(* CODESYS project NETWORK.library
   Author: OSCAT
   Version: 1.3.5.1
   Description: Oscat Network Version 07/2017 aus *.lib
      Formale Korrekturen von annD und Referenzen "Variabeln LOC_DT et.al." für Kompatibilität mit Codesys 3.5.16.0 angepasst
   Title: NETWORK
   Placeholder: OSCAT_NETWORK
   DefaultNamespace: OSCAT_NETWORK
   Company: OSCAT

Project tree, tasks and I/O mapping:
  libraries: IecSfc, 3.4.2.0 (System); Analyzation, 3.5.15.0 (System); Standard, 3.5.15.0 (System); BASIC, 3.5.16.0 (OSCAT); SysFile, 3.5.15.0 (System); SysSocket, 3.5.15.0 (System); SysSocket2, 3.5.16.10 (System); SysTypes Interfaces, 3.5.2.0 (System)
  Data types/
    DATA_LOG/
      data type DLOG_CRON_DATA
      data type DLOG_CRON_ELEMENT
      data type DLOG_DATA
      data type DLOG_REAL_ARRAY_DATA
      data type DLOG_REAL_ARRAY_ELEMENT
      data type DLOG_RETAIN
      data type DLOG_SAVE
      data type LOG_CONTROL
      data type PRINTF_DATA
      data type UNI_CIRCULAR_BUF
      data type UNI_CIRCULAR_BUFFER_DATA
      data type us_LOG_VIEWPORT
    DATABASE/
      data type MYSQL_COM
      data type MYSQL_INFO
    FILE_SERVER/
      data type FILE_PATH_DATA
      data type FILE_SERVER_DATA
      data type FILE_SERVER_RUNTIME_DATA
    NET_VAR/
      data type NET_VAR_DATA
    NETWORK/
      data type IP2GEO_DATA
      data type IP_C
      data type IP_FIFO_DATA
      data type NETWORK_BUFFER
      data type NETWORK_BUFFER_SHORT
      data type NW_BUF_LONG
      data type NW_BUF_SHORT
      data type URL
      data type VMAP_DATA
      data type XML_CONTROL
    TELNET_VISION/
      data type us_TN_INPUT_CONTROL
      data type us_TN_INPUT_CONTROL_DATA
      data type us_TN_MENU
      data type us_TN_MENU_POPUP
      data type us_TN_SCREEN
    WEATHER/
      data type WORLD_WEATHER_CUR
      data type WORLD_WEATHER_DATA
      data type WORLD_WEATHER_DAY
      data type YAHOO_WEATHER_DATA
      data type YAHOO_WEATHER_FORECAST_DAY
  Global Variables/
    global variables Constants
    global variables Globale_Variablen
  POUs/
    CONVERT/
      function block BASE64_DECODE_STR [ST]
      function block BASE64_DECODE_STREAM [ST]
      function block BASE64_ENCODE_STR [ST]
      function block BASE64_ENCODE_STREAM [ST]
      function HTML_DECODE [ST]
      function HTML_ENCODE [ST]
      function IP4_CHECK [ST]
      function IP4_DECODE [ST]
      function IP4_TO_STRING [ST]
      function IS_IP4 [ST]
      function IS_URLCHR [ST]
      function MD5_AUX [ST]
      function block MD5_CRAM_AUTH [ST]
      function block MD5_STR [ST]
      function block MD5_STREAM [ST]
      function MD5_TO_STRH [ST]
      function block RC4_CRYPT_STREAM [ST]
      function block SHA1_STR [ST]
      function block SHA1_STREAM [ST]
      function SHA1_TO_STRH [ST]
      function STRING_TO_URL [ST]
      function URL_DECODE [ST]
      function URL_ENCODE [ST]
      function URL_TO_STRING [ST]
    DATA_LOG/
      function block DLOG_BOOL [ST]
      function block DLOG_CRON_TAB [ST]
      function block DLOG_DINT [ST]
      function block DLOG_DT [ST]
      function block DLOG_FILE_TO_FTP [ST]
      function block DLOG_FILE_TO_SMTP [ST]
      function block DLOG_REAL [ST]
      function block DLOG_REAL_ARRAY [ST]
      function block DLOG_STORE_FILE_CSV [ST]
      function block DLOG_STORE_FILE_HTML [ST]
      function block DLOG_STORE_FILE_XML [ST]
      function block DLOG_STORE_MYSQL [ST]
      function block DLOG_STORE_RRD [ST]
      function block DLOG_STRING [ST]
    DATABASE/
      function block MYSQL_AUTH [ST]
      function block MYSQL_CONTROL [ST]
    DEMO/
      program BASE64_DEMO [CFC]
      program CSV_PARSER_BUF_DEMO [ST]
      program CSV_PARSER_FILE_DEMO [ST]
      program DLOG_FILE_CSV_DEMO [CFC]
      program DLOG_FILE_CSV_FTP_DEMO [CFC]
      program DLOG_FILE_CSV_SMTP_DEMO [CFC]
      program DLOG_FILE_HTML_DEMO [CFC]
      program DLOG_FILE_XML_DEMO [CFC]
      program DLOG_MYSQL_DEMO [CFC]
      program DLOG_RRD_DEMO [CFC]
      program DNS_DYN_DEMO [CFC]
      program DNS_REV_DEMO [CFC]
      program DNS_SNTP_SYSLOG_DEMO [CFC]
      program FILE_BLOCK_DEMO [CFC]
      program FTP_CLIENT_DEMO [CFC]
      program GET_WAN_IP_DEMO [CFC]
      program HTTP_DEMO [CFC]
      program INI_PARSER_BUF_DEMO [ST]
      program INI_PARSER_FILE_DEMO [ST]
      program IP2GEO_DEMO [CFC]
      program IRTRANS_DEMO [CFC]
      program MB_CLIENT_DEMO [CFC]
      program MB_SERVER_DEMO [CFC]
      program MD5_CRAM_AUTH_DEMO [CFC]
      program NET_VAR_MASTER_DEMO [CFC]
      program NET_VAR_SLAVE_DEMO [CFC]
      program RC4_CRYPT_DEMO [CFC]
      program SHA1_MD5_DEMO [CFC]
      program SMTP_CLIENT_DEMO [CFC]
      program SPIDER_DEMO [CFC]
      program TELNET_LOG_DEMO [CFC]
      program TELNET_PRINT_DEMO [CFC]
      program TN_VISION_DEMO_1 [ST]
      program TN_VISION_DEMO_2 [ST]
      program WORLD_WEATHER_DEMO [CFC]
      program YAHOO_WEATHER_DEMO [CFC]
    DRIVER/
      function block IRTRANS_DECODE [ST]
      function block IRTRANS_RCV_1 [ST]
      function block IRTRANS_RCV_4 [ST]
      function block IRTRANS_RCV_8 [ST]
      function block IRTRANS_SERVER [ST]
      function block IRTRANS_SND_1 [ST]
      function block IRTRANS_SND_4 [ST]
      function block IRTRANS_SND_8 [ST]
    FILE/
      function block CSV_PARSER_BUF [ST]
      function block CSV_PARSER_FILE [ST]
      function block FILE_BLOCK [ST]
      function FILE_PATH_SPLIT [ST]
      function block INI_PARSER_BUF [ST]
      function block INI_PARSER_FILE [ST]
    HARDWARE/
      function block FILE_SERVER [ST]
      function block FILE_SERVER_RUNTIME [ST]
      function block IP_CONTROL2 [ST]
      function block IP_CONTROL [ST]
    NET_VAR/
      function block NET_VAR_BOOL8 [ST]
      function block NET_VAR_BUFFER [ST]
      function block NET_VAR_CONTROL [ST]
      function block NET_VAR_DWORD8 [ST]
      function block NET_VAR_REAL8 [ST]
      function block NET_VAR_STRING [ST]
      function block NET_VAR_X8 [ST]
    NETWORK/
      function block DNS_CLIENT [ST]
      function block DNS_DYN [ST]
      function block DNS_REV_CLIENT [ST]
      function block FTP_CLIENT [ST]
      function block GET_WAN_IP [ST]
      function block HTTP_GET [ST]
      function block IP2GEO [ST]
      function block MB_CLIENT [ST]
      function block MB_SERVER [ST]
      function block MB_SERVER_1 [ST]
      function block MB_VMAP [ST]
      function block READ_HTTP [ST]
      function block SMTP_CLIENT [ST]
      function block SNTP_CLIENT [ST]
      function block SNTP_SERVER [ST]
      function block SPIDER_ACCESS [ST]
      function block SYS_LOG [ST]
      function block TELNET_LOG [ST]
      function block TELNET_PRINT [ST]
    OTHER/
      function ELEMENT_COUNT [ST]
      function ELEMENT_GET [ST]
      function block IP_FIFO [ST]
      function block LOG_MSG [ST]
      function block LOG_VIEWPORT [ST]
      function NETWORK_VERSION [ST]
      function block PRINT_SF [ST]
      function block UNI_CIRCULAR_BUFFER [ST]
      function block XML_READER [ST]
    TELNET_VISION/
      function block TN_FRAMEWORK [ST]
      function block TN_INPUT_CONTROL [ST]
      function block TN_INPUT_EDIT_LINE [ST]
      function block TN_INPUT_MENU_BAR [ST]
      function block TN_INPUT_MENU_POPUP [ST]
      function block TN_INPUT_SELECT_POPUP [ST]
      function block TN_INPUT_SELECT_TEXT [ST]
      function block TN_RECEIVE [ST]
      function block TN_SC_ADD_SHADOW [ST]
      function block TN_SC_AREA_RESTORE [ST]
      function block TN_SC_AREA_SAVE [ST]
      function block TN_SC_BOX [ST]
      function block TN_SC_FILL [ST]
      function block TN_SC_LINE [ST]
      function block TN_SC_READ_ATTR [ST]
      function block TN_SC_READ_CHAR [ST]
      function TN_SC_SHADOW_ATTR [ST]
      function block TN_SC_VIEWPORT [ST]
      function block TN_SC_WRITE [ST]
      function block TN_SC_WRITE_ATTR [ST]
      function block TN_SC_WRITE_C [ST]
      function block TN_SC_WRITE_CHAR [ST]
      function block TN_SC_WRITE_EOS [ST]
      function TN_SC_XY2_ERROR [ST]
      function TN_SC_XY_ERROR [ST]
      function block TN_SEND_ROWS [ST]
    WEATHER/
      function block MOON_PHASE [ST]
      function block WORLD_WEATHER [ST]
      function block WORLD_WEATHER_DESC_GE [ST]
      function block WORLD_WEATHER_ICON_OSCAT [ST]
      function block YAHOO_WEATHER [ST]
      function block YAHOO_WEATHER_DESC_GE [ST]
      function block YAHOO_WEATHER_ICON_OSCAT [ST]
*)

// Data types/DATA_LOG/DLOG_CRON_DATA
TYPE DLOG_CRON_DATA :
STRUCT
	CE : ARRAY [0..5] OF DLOG_CRON_ELEMENT;
END_STRUCT
END_TYPE

// Data types/DATA_LOG/DLOG_CRON_ELEMENT
TYPE DLOG_CRON_ELEMENT :
STRUCT
	ELEMENTS : ARRAY [0..59] OF BOOL;
	VALUE : INT;
	VALUE_MIN : INT;
	VALUE_MAX : INT;
	ALL_SELECTED : BOOL;
END_STRUCT
END_TYPE

// Data types/DATA_LOG/DLOG_DATA
TYPE DLOG_DATA :
STRUCT
	STORE_TYPE : BYTE;
	ADD_COM : INT;
	ADD_DATA_REQ : BOOL;
	CLOCK_TRIG : BOOL;
	ID_MAX : USINT;
	DTI : DT;
	UCB : UNI_CIRCULAR_BUFFER_DATA;
	LOAD_TIME_MAX : TIME;
	NEW_FILE : STRING;
	NEW_FILE_SIZE : UDINT;
	NEW_FILE_RTRIG : BOOL;
END_STRUCT
END_TYPE

// Data types/DATA_LOG/DLOG_REAL_ARRAY_DATA
TYPE
	DLOG_REAL_ARRAY_DATA : ARRAY [1..64] OF DLOG_REAL_ARRAY_ELEMENT;
END_TYPE

// Data types/DATA_LOG/DLOG_REAL_ARRAY_ELEMENT
TYPE DLOG_REAL_ARRAY_ELEMENT :
STRUCT
	VALUE : REAL;
	DELTA : REAL;
	COLUMN : STRING(10);
	_DELTA_LAST : 	REAL;
	_VALUE_LAST : 	REAL;
END_STRUCT
END_TYPE

// Data types/DATA_LOG/DLOG_RETAIN
TYPE DLOG_RETAIN :
STRUCT
	FN_REM : STRING;
	COLOR : BOOL;
	HEAD: BOOL;
	TRIG_CNT : UDINT;
	TRIG_CNT_TOTAL : UDINT;
END_STRUCT
END_TYPE

// Data types/DATA_LOG/DLOG_SAVE
TYPE DLOG_SAVE :
STRUCT
	FN_REM : STRING;
	COLOR : BOOL;
	HEAD: BOOL;
	TRIG_CNT : UDINT;
	TRIG_CNT_TOTAL : UDINT;
END_STRUCT
END_TYPE

// Data types/FILE_SERVER/FILE_PATH_DATA
TYPE FILE_PATH_DATA :
STRUCT
	DRIVE : STRING(3);
	DIRECTORY : STRING(OSCAT_BASIC.STRING_LENGTH);
	FILENAME : STRING;
END_STRUCT
END_TYPE

// Data types/FILE_SERVER/FILE_SERVER_DATA
TYPE FILE_SERVER_DATA :
STRUCT
	FILE_OPEN : BOOL;
	FILENAME : STRING;
	MODE : BYTE;
	OFFSET : UDINT;
	FILE_SIZE : UDINT;
	ERROR : BYTE;
	RUNTIME : FILE_SERVER_RUNTIME_DATA;
END_STRUCT
END_TYPE

// Data types/FILE_SERVER/FILE_SERVER_RUNTIME_DATA
TYPE FILE_SERVER_RUNTIME_DATA :
STRUCT
	TIME_FILE_OPEN_CUR : UDINT;
	TIME_FILE_OPEN_MAX : UDINT;
	TIME_FILE_OPEN_MIN : UDINT;
	TIME_FILE_CLOSE_CUR : UDINT;
	TIME_FILE_CLOSE_MAX : UDINT;
	TIME_FILE_CLOSE_MIN : UDINT;
	TIME_FILE_READ_CUR: UDINT;
	TIME_FILE_READ_MAX : UDINT;
	TIME_FILE_READ_MIN : UDINT;
	TIME_FILE_WRITE_CUR : UDINT;
	TIME_FILE_WRITE_MAX : UDINT;
	TIME_FILE_WRITE_MIN : UDINT;
	TIME_FILE_SEEK_CUR : UDINT;
	TIME_FILE_SEEK_MAX : UDINT;
	TIME_FILE_SEEK_MIN : UDINT;
	TIME_FILE_TELL_CUR : UDINT;
	TIME_FILE_TELL_MAX : UDINT;
	TIME_FILE_TELL_MIN : UDINT;
	TIME_FILE_DELETE_CUR : UDINT;
	TIME_FILE_DELETE_MAX : UDINT;
	TIME_FILE_DELETE_MIN : UDINT;
END_STRUCT
END_TYPE

// Data types/NETWORK/IP2GEO_DATA
TYPE IP2GEO_DATA :
STRUCT
	STATE : BOOL;
	IP4 : DWORD;
	COUNTRY_CODE : STRING(2);
	COUNTRY_NAME : STRING(20);
	REGION_CODE : STRING(2);
	REGION_NAME : STRING(20);
	CITY : STRING(20);
	GEO_LATITUDE : REAL;
	GEO_LONGITUDE : REAL;
	TIME_ZONE_NAME : STRING(20);
	GMT_OFFSET : INT;
	IS_DST : BOOL;
END_STRUCT
END_TYPE

// Data types/NETWORK/IP_C
TYPE IP_C :
STRUCT
	C_MODE : BYTE;						(*W Mode: TCP/UCP AKTIV/PASSIV                               *)
	C_PORT : WORD;						(*W Portnummer                                               *)
	C_IP : DWORD;						(*W IP-Adresse gepackt wwxxyyzz = www.xxx.yyy.zzz            *)
	C_STATE : BYTE;						(*R Verbindungsstatus ON/OFF + Flanke ON/OFF                 *)
	C_ENABLE : BOOL;					(*W Freigabe für Connect                                     *)
	R_OBSERVE : BOOL;					(*W Empfang ueberwachen                                      *)
	TIME_RESET : BOOL;					(*W Alle Timer ruecksetzen                                   *)
	ERROR : DWORD;					(*R vvwwxxyy (vv = CON_ERROR, ww = SEN_ERROR, xx = REC_ERROR *)
	FIFO : IP_FIFO_DATA;					(*I IP FIFO Struktur                                         *)
	MAILBOX : ARRAY [1..16] OF BYTE;	(*I Mailbox: Datenbereich für Bausteindatenaustausch         *)
	ResultSend:RTS_IEC_RESULT; 			(*Result of TCP Send call*)
	ResultReceive:RTS_IEC_RESULT;		(*Result of TCP Receive call*)
END_STRUCT
END_TYPE

// Data types/NETWORK/IP_FIFO_DATA
TYPE IP_FIFO_DATA :
STRUCT
	X : ARRAY [1..128] OF BYTE; 	(* IP_ID FIFO Speicher          *)
	Y : ARRAY [1..128] OF BYTE; 	(* IP_ID Zähler                 *)
	ID : BYTE;					(* höchste vergabene id         *)
	MAX_ID : BYTE;				(* maximal Anmeldungen pro ID   *)
	INIT : BOOL;					(* Initialisierung durchgeführt *)
	EMPTY : BOOL;				(* FIFO leer                    *)
	FULL : BOOL;					(* FIFO voll                    *)
	TOP : INT;					(* maximale anzahl in FIFO      *)
	NW : INT;					(* Schreibzeiger                *)
	NR : INT;						(* Lesezeiger                   *)
END_STRUCT
END_TYPE

// Data types/DATA_LOG/LOG_CONTROL
TYPE LOG_CONTROL :
STRUCT
	NEW_MSG : STRING(LOG_SIZE); (* neue Nachricht für den Datenbuffer *)
	NEW_MSG_OPTION : DWORD;
	LEVEL : BYTE;
	SIZE : INT := LOG_MAX; (* Anzahl der Strings im LOG_DATA *)
	RESET : BOOL; (* Nachrichtenbuffer löschen *)
	PRINTF : PRINTF_DATA; (* Array PRINTF Parameter *)
	MSG : ARRAY [0..LOG_MAX] OF STRING(LOG_SIZE); (* Array Message *)
	MSG_OPTION : ARRAY [0..LOG_MAX] OF DWORD; (* Array Options *)
	UPDATE_COUNT : UINT; (* Updatezähler *)
	IDX : INT; (* aktueller Nachrichten-Index *)
	RING_MODE : BOOL; (* Bufferüberlauf erkannt *)
END_STRUCT
END_TYPE

// Data types/DATABASE/MYSQL_COM
TYPE MYSQL_COM :
STRUCT
	S_BUF : NETWORK_BUFFER;
	R_BUF : NETWORK_BUFFER;
	SQL_CON : BOOL;
	SQL_URL : STRING(OSCAT_BASIC.STRING_LENGTH);
	SQL_PACKET_NO : BYTE;
	TIMEOUT : TIME;
	DNS_IP4 : DWORD;
	SQL_RCV_STATE : BYTE;
	ERROR_C : DWORD;
	ERROR_T : BYTE;
END_STRUCT
END_TYPE

// Data types/DATABASE/MYSQL_INFO
TYPE MYSQL_INFO :
STRUCT
	SERVER_PROTOCOL_VERSION : BYTE;
	SERVER_CAPABILITIES : WORD;
	SERVER_STATUS : WORD;
	SERVER_LANGUAGE : BYTE;
	SQL_CONNECTED : BOOL;
	SQL_ERROR : STRING(OSCAT_BASIC.STRING_LENGTH);
	DATA_INSERT_AKTIV : BOOL;
	DATA_INSERT_OK_CNT : UDINT;
	DATA_INSERT_NOK_CNT : UDINT;
END_STRUCT
END_TYPE

// Data types/NET_VAR/NET_VAR_DATA
TYPE NET_VAR_DATA :
STRUCT
	CYCLE : UDINT;
	STATE : BYTE;
	INDEX : INT;
	ID_MAX : USINT;
	ERROR_ID : BYTE;
	BUF_SIZE : UINT;
	S_BUF : NETWORK_BUFFER;
	R_BUF : NETWORK_BUFFER;
END_STRUCT
END_TYPE

// Data types/NETWORK/NETWORK_BUFFER
TYPE NETWORK_BUFFER :
STRUCT
	SIZE : UINT;
	BUFFER : NW_BUF_LONG;
END_STRUCT
END_TYPE

// Data types/NETWORK/NETWORK_BUFFER_SHORT
TYPE NETWORK_BUFFER_SHORT :
STRUCT
	SIZE : UINT;
	BUFFER : NW_BUF_SHORT;
END_STRUCT
END_TYPE

// Data types/NETWORK/NW_BUF_LONG
TYPE
	NW_BUF_LONG  : ARRAY[0..NETWORK_BUFFER_LONG_SIZE] OF BYTE;
END_TYPE

// Data types/NETWORK/NW_BUF_SHORT
TYPE
	NW_BUF_SHORT : ARRAY[0..NETWORK_BUFFER_SHORT_SIZE] OF BYTE;
END_TYPE

// Data types/DATA_LOG/PRINTF_DATA
TYPE PRINTF_DATA : ARRAY [1..11]  OF STRING(LOG_SIZE);
END_TYPE

// Data types/DATA_LOG/UNI_CIRCULAR_BUF
TYPE
	UNI_CIRCULAR_BUF : ARRAY [0..8191] OF BYTE;
END_TYPE

// Data types/DATA_LOG/UNI_CIRCULAR_BUFFER_DATA
TYPE UNI_CIRCULAR_BUFFER_DATA :
STRUCT
	D_MODE : INT;
	D_SIZE : INT;
	D_HEAD : WORD;
	D_STRING : STRING(OSCAT_BASIC.STRING_LENGTH);
	D_REAL : REAL;
	D_DWORD : DWORD;
	BUF_SIZE : UINT;
	BUF_COUNT : UINT;
	BUF_USED : USINT;
	BUF_USED_MAX : USINT;
	BUF_DATA_CNT : UDINT;
	BUF_DATA_LOST : UDINT;
	BUF : UNI_CIRCULAR_BUF;
	_GetStart : UINT;
	_GetEnd : UINT;
	_Last : UINT;
	_First : UINT;
END_STRUCT
END_TYPE

// Data types/NETWORK/URL
TYPE URL :
STRUCT
	PROTOCOL : STRING(10);
	USER : STRING(32);
	PASSWORD : STRING(32);
	DOMAIN : STRING(80);
	PORT : WORD;
	PATH : STRING(80);
	QUERY : STRING(OSCAT_BASIC.STRING_LENGTH);
	ANCHOR : STRING(40);
	HEADER : STRING(160);
END_STRUCT
END_TYPE

// Data types/DATA_LOG/us_LOG_VIEWPORT
TYPE us_LOG_VIEWPORT :
STRUCT
	LINE_ARRAY : ARRAY [1..40] OF INT;
	COUNT : INT; (* Anzahl der sichtbaren Nachtrichten *)
	UPDATE_COUNT : UINT; (* Updatezähler *)
	MOVE_TO_X : INT; (* Steuerung der Nachrichtenanzeige *)
	UPDATE : BOOL; (* Daten wurden geändert -> neuzeichnen *)
END_STRUCT
END_TYPE

// Data types/TELNET_VISION/us_TN_INPUT_CONTROL
TYPE us_TN_INPUT_CONTROL :
STRUCT
	bo_Enable: BOOL; (* Bearbeitung freigeben/sperren *)
	bo_Update_all: BOOL; (* All Elemente neu zeichnen *)
	bo_Reset_Fokus: BOOL; (* Fokus auf 1. Element setzen *)
	in_Focus_at: INT; (* Controlelement mit aktivem Fokus *)
	in_Count: INT; (* Anzahl der benutzen Control-Elemente *)
	in_ToolTip_X: INT; (* Tooltip Text X-Offset *)
	in_ToolTip_Y: INT; (* Tooltip Text Y-Offset *)
	by_ToolTip_Attr: BYTE; (* Tooltip Text Attribute *)
	in_ToolTip_Size: INT; (* Tooltip Text länge *)
	usa_TN_INPUT_CONTROL_DATA: ARRAY [1..20] OF us_TN_INPUT_CONTROL_DATA;
END_STRUCT
END_TYPE

// Data types/TELNET_VISION/us_TN_INPUT_CONTROL_DATA
TYPE us_TN_INPUT_CONTROL_DATA :
STRUCT
 	by_Input_Exten_Code: BYTE;
	by_Input_ASCII_Code: BYTE;
	bo_Input_ASCII_IsNum: BOOL;
	in_Title_X_Offset: INT; (* Title Text X-Offset *)
	in_Title_Y_Offset: INT; (* Title Text Y-Offset *)
	by_Title_Attr: BYTE; (* Title Text Attribute *)
	st_Title_String: STRING; (* Title Text String *)
	in_Cursor_X: INT; (* aktuelle Cursor X-Position *)
	in_Cursor_Y: INT; (* aktuelle Cursor Y-Position *)
	in_Type: INT; (* Type des Elements *)
	in_X: INT; (* Element X-Position *)
	in_Y: INT; (* Element Y-Position *)
	in_Cursor_Pos: INT; (* aktuelle Cursorposition *)
	by_Attr_mF: BYTE; (* Text Attribute mit Fokus *)
	by_Attr_oF: BYTE; (* Text Attribute ohne Fokus *)
	in_selected: INT; (* Text Item wurde ausgewählt *)
	st_Input_Mask: STRING; (* Text Eingabemaske *)
	st_Input_Data: STRING(OSCAT_BASIC.STRING_LENGTH); (* Text aktuelle Eingabedaten *)
	st_Input_String: STRING; (* Text Kopie nach Return-Taste *)
	st_Input_ToolTip: STRING; (* Text ToolTip (Eingabeinformation) *)
	in_Input_Option: INT; (* Text Ausgabe-Optionen *)
	bo_Input_Entered: BOOL; (* RETURN-Taste wurde betätigt *)
	bo_Input_Hidden: BOOL; (* Text versteckete Eingabe mit '*' *)
	bo_Input_Only_Num: BOOL; (* Text nur Nummerneingabe zulassen *)
	bo_Focus: BOOL; (* Element besitzt den Fokus *)
	bo_Update_Input: BOOL; (* Element wegen Benutzereingabe neuzeichnen *)
	bo_Update_All: BOOL; (* Element komplett neuzeichnen *)

END_STRUCT
END_TYPE

// Data types/TELNET_VISION/us_TN_MENU
TYPE us_TN_MENU :
STRUCT
	st_Menu_Text: STRING(OSCAT_BASIC.STRING_LENGTH); (* X Menue Texte *)
	in_Menu_E_Count: INT; (* Menue Elemente Anzahl *)
	in_Y: INT; (* Menue Zeilennummer  Y-Position *)
	in_X: INT; (* Menue Spaltennummer X-Position *)
	by_Attr_mF: BYTE; (* Text Attribute mit Fokus *)
	by_Attr_oF: BYTE; (* Text Attribute ohne Fokus *)
	in_X_SM_new: INT; (* neue Sub-Menu X-Position *)
	in_Y_SM_new: INT; (* neue Sub-Menu Y-Position *)
	in_X_SM_old: INT; (* alte Sub-Menu X-Position *)
	in_Y_SM_old: INT; (* alte Sub-Menu Y-Position *)
	in_Cur_Menu_Item: INT; (* aktuelles Haupt-Menue *)
	in_Cur_Sub_Item: INT; (* aktuelles Sub-Menue *)
	in_State: INT; (*   Menu status   *)
	in_Menu_Selected: INT; (* X Menu-Item mit Enter angewwählt *)
	bo_Create: BOOL; (* X Menu erzeugen *)
	bo_Destroy: BOOL; (* X Menu entfernen *)
	bo_Update: BOOL; (* X Menu updaten *)
END_STRUCT
END_TYPE

// Data types/TELNET_VISION/us_TN_MENU_POPUP
TYPE us_TN_MENU_POPUP :
STRUCT
	st_Menu_Text: STRING(OSCAT_BASIC.STRING_LENGTH); (* X Menue Texte *)
	in_Menu_E_Count: INT; (* Menue Elemente Anzahl *)
	in_X: INT; (* X Menue X-Position *)
	in_Y: INT; (* X Menue Y-Position *)
	in_Cols: INT; (* Menue Spaltenanzahl *)
	in_Rows: INT; (* Menue Zeilenanzahl *)
	in_Cur_Item: INT; (* X aktuelles Sub-Menue *)
	by_Attr_mF: BYTE; (* X Text Attribute mit Fokus	*)
	by_Attr_oF: BYTE; (* X Text Attribute ohne Fokus *)
	by_Input_Exten_Code: BYTE; (* X Tastencode: Sondertasten *)
	bo_Create: BOOL; (* X Popup-Menu erzeugen *)
	bo_Destroy: BOOL; (* X Popup-Menu entfernen *)
	bo_Update: BOOL; (* X Popup-Menu updaten *)
	bo_Activ: BOOL; (*   Popup-Menu ist aktiv *)
END_STRUCT
END_TYPE

// Data types/TELNET_VISION/us_TN_SCREEN
TYPE us_TN_SCREEN :
STRUCT
	bya_CHAR: ARRAY [0..1919] OF BYTE;
	bya_COLOR: ARRAY [0..1919] OF BYTE;
	bya_BACKUP: ARRAY [0..1919] OF BYTE;
	bya_Line_Update: ARRAY [0..23] OF BOOL;
	by_Input_Exten_Code: BYTE;
	by_Input_ASCII_Code: BYTE;
	bo_Input_ASCII_IsNum: BOOL;
	in_Page_Number: INT; (* aktive Seiten-Nr. *)
	in_Cursor_X: INT; (* Cursor X-Position *)
	in_Cursor_Y: INT; (* Cursor Y-Position *)
	in_EOS_Offset: INT; (* End of String Offset *)
	by_Clear_Screen_Attr: BYTE; (* Clear-Screen Attr *)
	bo_Clear_Screen: BOOL; (* Clear-Screen auslösen *)
	bo_Modal_Dialog: BOOL; (* Modaler Dialog ist aktiv *)
	bo_Menue_Bar_Dialog: BOOL; (* Menue Dialog ist aktiv *)
END_STRUCT
END_TYPE

// Data types/NETWORK/VMAP_DATA
TYPE VMAP_DATA :
STRUCT
	FC : DWORD;
	V_ADR : INT;
	V_SIZE : INT;
	P_ADR : INT;
	TIME_OUT : TIME;
END_STRUCT
END_TYPE

// Data types/WEATHER/WORLD_WEATHER_CUR
TYPE WORLD_WEATHER_CUR :
STRUCT
	OBSERVATION_TIME : STRING(8);
	TEMP_C : INT;
	WEATHER_CODE : INT;
	WEATHER_DESC : STRING(60);
	WEATHER_ICON : INT;
	WIND_SPEED_MILES : INT;
	WIND_SPEED_KMPH : INT;
	WIND_DIR_DEGREE : INT;
	WIND_DIR16POINT : STRING(3);
	PRECIPMM : REAL;
	HUMIDITY : INT;
	VISIBILITY : INT;
	PRESSURE : INT;
	CLOUDOVER : INT;
END_STRUCT
END_TYPE

// Data types/WEATHER/WORLD_WEATHER_DATA
TYPE WORLD_WEATHER_DATA :
STRUCT
	CUR : WORLD_WEATHER_CUR;
	DAY : ARRAY [0..4] OF WORLD_WEATHER_DAY;
END_STRUCT
END_TYPE

// Data types/WEATHER/WORLD_WEATHER_DAY
TYPE WORLD_WEATHER_DAY :
STRUCT
	DATE_OF_DAY : STRING(10);
	TEMP_MAX_C : INT;
	TEMP_MAX_F : INT;
	TEMP_MIN_C : INT;
	TEMP_MIN_F : INT;
	WIND_SPEED_MILES : INT;
	WIND_SPEED_KMPH : INT;
	WIND_DIR_DEGREE : INT;
	WIND_DIR16POINT : STRING(3);
	WEATHER_CODE : INT;
	WEATHER_DESC : STRING(60);
	WEATHER_ICON : INT;
	PRECIPMM : REAL;
END_STRUCT
END_TYPE

// Data types/NETWORK/XML_CONTROL
TYPE XML_CONTROL :
STRUCT
	COMMAND : WORD;
	WATCHDOG : TIME;
	START_POS : UINT;
	STOP_POS : UINT;
	COUNT : UINT;
	TYP : INT;
	LEVEL : UINT;
	PATH : STRING(OSCAT_BASIC.STRING_LENGTH);
	ELEMENT : STRING(OSCAT_BASIC.STRING_LENGTH);
	ATTRIBUTE : STRING(OSCAT_BASIC.STRING_LENGTH);
	VALUE : STRING(OSCAT_BASIC.STRING_LENGTH);
	BLOCK1_START : UINT;
	BLOCK1_STOP : UINT;
	BLOCK2_START : UINT;
	BLOCK2_STOP : UINT;
END_STRUCT
END_TYPE

// Data types/WEATHER/YAHOO_WEATHER_DATA
TYPE YAHOO_WEATHER_DATA :
STRUCT
	LOCATION_CITY : STRING(40);   					(* THE LOCATION OF THIS FORECAST: CITY: CITY NAME  *)
	LOCATION_REGION : STRING(20);   					(* THE LOCATION OF THIS FORECAST: REGION: STATE, TERRITORY, OR REGION, IF GIVEN *)
	LOCATION_COUNTRY : STRING(20);   				(* THE LOCATION OF THIS FORECAST: COUNTRY: TWO-CHARACTER COUNTRY CODE *)
	UNIT_TEMPERATURE : STRING(1);    				(* TEMPERATURE: DEGREE UNITS, F FOR FAHRENHEIT OR C FOR CELSIUS *)
	UNIT_DISTANCE : STRING(2);    					(* DISTANCE: UNITS FOR DISTANCE, MI FOR MILES OR KM FOR KILOMETERS *)
	UNIT_PRESSURE : STRING(2);    					(* PRESSURE: UNITS OF BAROMETRIC PRESSURE, IN FOR POUNDS PER SQUARE INCH OR MB FOR MILLIBARS *)
	UNIT_SPEED : STRING(4);    						(* SPEED: UNITS OF SPEED, MPH FOR MILES PER HOUR OR KPH FOR KILOMETERS PER HOUR *)
	WIND_CHILL : INT;              							(* FORECAST INFORMATION ABOUT WIND CHILL IN DEGREES *)
	WIND_DIRECTION : INT;              						(* FORECAST INFORMATION ABOUT WIND DIRECTION, IN DEGREES *)
	WIND_SPEED : REAL;             						(* FORECAST INFORMATION ABOUT WIND SPEED, IN THE UNITS (MPH OR KPH)*)
	ATMOSPHERE_HUMIDITY : INT;              				(* FORECAST INFORMATION ABOUT CURRENT ATMOSPHERIC HUMIDITY: HUMIDITY, IN PERCENT  *)
	ATMOSPHERE_PRESSURE : REAL;             			(* FORECAST INFORMATION ABOUT CURRENT ATMOSPHERIC PRESSURE: BAROMETRIC PRESSURE, IN THE UNITS (IN OR MB) *)
	ATMOSPHERE_VISIBILITY : REAL;             			(* FORECAST INFORMATION ABOUT CURRENT ATMOSPHERIC VISIBILITY, IN THE UNITS (MI OR KM) *)
	ATMOSPHERE_RISING : INT;              					(* FORECAST INFORMATION ABOUT RISING: STATE OF THE BAROMETRIC PRESSURE: STEADY (0), RISING (1), OR FALLING (2). (INTEGER: 0, 1, 2) *)
	ASTRONOMY_SUNRISE : STRING(10);   				(* SUNRISE: TODAY'S SUNRISE TIME. THE TIME IS A STRING IN A LOCAL TIME FORMAT OF "H:MM AM/PM" *)
	ASTRONOMY_SUNSET : STRING(10);   				(* SUNSET: TODAY'S SUNSET TIME. THE TIME IS A STRING IN A LOCAL TIME FORMAT OF "H:MM AM/PM", *)
	GEO_LATITUDE : REAL;             						(* THE LATITUDE OF THE LOCATION *)
	GEO_LONGITUDE : REAL;             					(* THE LONGITUDE OF THE LOCATION *)
	CUR_CONDITIONS_TEMP : INT;              				(* THE CURRENT WEATHER CONDITIONS: TEMP: THE CURRENT TEMPERATURE, IN THE UNITS (F OR C) *)
	CUR_CONDITIONS_TEXT : STRING(40);   			(* THE CURRENT WEATHER CONDITIONS: TEXT: A TEXTUAL DESCRIPTION OF CONDITIONS *)
	CUR_CONDITIONS_CODE : INT;              				(* THE CURRENT WEATHER CONDITIONS: CODE: THE CONDITION CODE FOR THIS FORECAST *)
	CUR_CONDITIONS_ICON : INT;			  			(* THE CURRENT WEATHER CONDITIONS: ICON: THE CONDITION ICON FOR THIS FORECAST *)
	FORECAST_TODAY_LOW_TEMP : INT;              		(* THE FORECAST TODAY WEATHER CONDITIONS: THE FORECASTED LOW TEMPERATURE FOR THIS DAY IN THE UNITS (F OR C) *)
	FORECAST_TODAY_HIGH_TEMP : INT;              		(* THE FORECAST TODAY WEATHER CONDITIONS: THE FORECASTED HIGH TEMPERATURE FOR THIS DAY IN THE UNITS (F OR C) *)
	FORECAST_TODAY_TEXT : STRING(40);   			(* THE FORECAST TODAY WEATHER CONDITIONS: TEXT: A TEXTUAL DESCRIPTION OF CONDITIONS *)
	FORECAST_TODAY_CODE : INT;              				(* THE CURRENT WEATHER CONDITIONS: CODE: THE CONDITION CODE FOR THIS FORECAST *)
	FORECAST_TODAY_ICON : INT;			  		(* THE CURRENT WEATHER CONDITIONS: ICON: THE CONDITION ICON FOR THIS FORECAST *)
	FORECAST_TODAY_DATE_LONG : STRING(20);	  	(* THE CURRENT WEATHER CONDITIONS: DATE: DATE OF THE DAY *)
	FORECAST_DAY : ARRAY [1..9] OF YAHOO_WEATHER_FORECAST_DAY;	 (* THE CURRENT WEATHER DAYS ARRAY *)
END_STRUCT
END_TYPE

// Data types/WEATHER/YAHOO_WEATHER_FORECAST_DAY
TYPE YAHOO_WEATHER_FORECAST_DAY :
STRUCT
	LOW_TEMP : INT;					(* THE FORECAST WEATHER CONDITIONS: THE FORECASTED LOW TEMPERATURE FOR THIS DAY IN THE UNITS (F OR C) *)
	HIGH_TEMP : INT;              			(* THE FORECAST WEATHER CONDITIONS: THE FORECASTED HIGH TEMPERATURE FOR THIS DAY IN THE UNITS (F OR C) *)
	TEXT : STRING(40);   				(* THE FORECAST WEATHER CONDITIONS: TEXT: A TEXTUAL DESCRIPTION OF CONDITIONS *)
	DATE_LONG : STRING(20);   		(* THE FORECAST WEATHER CONDITIONS: DATE: DATE OF THE DAY *)
	CODE : INT;              				(* THE FORECAST WEATHER CONDITIONS: CODE: THE CONDITION CODE FOR THIS FORECAST *)
	ICON : INT;			  			(* THE FORECAST WEATHER CONDITIONS: ICON: THE CONDITION ICON FOR THIS FORECAST *)
END_STRUCT
END_TYPE

// Global Variables/Constants
VAR_GLOBAL CONSTANT
	NETWORK_BUFFER_LONG_SIZE : UINT := 4095;
	NETWORK_BUFFER_SHORT_SIZE : UINT := 1407;
	LOG_MAX : INT := 40;
	LOG_SIZE : INT := 80;
	ELEMENT_LENGTH : INT := 250;
END_VAR

// Global Variables/Globale_Variablen
VAR_GLOBAL
	(* ------- only for Beckhoff - TwinCat  --------- *)
	TCP_SERVER_RESET : BYTE; (* only for internaly use - do't modify *)
	sSrvNetId : STRING(23) := ''; (* String containing the network address of the TwinCAT TCP/IP Connection Server (e.g. '1.1.1.2.7.1'). For the local computer (default) an empty string may be specified *)
	sLocalHost : STRING(15) := ''; (* The local IP address (Ipv4) of the UDP client/server socket as a string (e.g. '172.33.5.1'). An empty string may be specified for the default network adapter *)
	(* --------------------------------------------- *)

	(* ------- only for CoDeSys --------------------        *)
	(* Configuration for SysLibSocket.lib                   *)
    (* Bit 0 = 1 -> PLCWinNT                                *)
    (* Bit 1 = 1 -> PLC WAGO 750-841                        *)
    (* Bit 2 = 1 -> PLC WAGO 750-881                        *)
	SYSLIBSOCKETS_OPTION : BYTE := BYTE#2#0000_0000;
	(* ---------------------------------------------------- *)

	LOG_CL : LOG_CONTROL;
END_VAR

// POUs/CONVERT/BASE64_DECODE_STR
FUNCTION_BLOCK BASE64_DECODE_STR
VAR_INPUT
	RUN : BOOL;
END_VAR
VAR_OUTPUT
	DONE : BOOL;
END_VAR
VAR_IN_OUT
	STR1 : STRING(192);
	STR2 : STRING(144);
END_VAR
VAR
	BASE64_DECODE_STREAM : BASE64_DECODE_STREAM;
	run_last : BOOL;
	buf1 : ARRAY [0..63] OF BYTE;
	buf2 : ARRAY [0..47] OF BYTE;
	mode : INT;
	size1 : INT;
	size2 : INT;
	end : INT;
	pos : INT;
END_VAR

(*
version 1.0	06. dec. 2009
programmer 	ks
tested by	ks

BASE64_DECODE_STR konvertiert einen BASE64 kodierten String in einen normalen String. 

*)

CASE mode OF
0:	IF RUN AND NOT run_last THEN
		DONE := FALSE;
		mode := 1;
		end := LEN(STR1);
		pos := 0;
		STR2 := '';
	END_IF;
1:
	size1 := MIN(48,end - pos);
	IF size1 > 0 THEN
		OSCAT_BASIC._STRING_TO_BUFFER(STR:=MID(STR1, size1, pos + 1), POS:=0, PT:=ADR(buf1), SIZE:=SIZEOF(buf1));
		BASE64_DECODE_STREAM(BUF1:=buf1 ,BUF2:=buf2 ,SIZE1:=size1 ,SIZE2=>size2);
		STR2 := CONCAT(STR2,OSCAT_BASIC.BUFFER_TO_STRING(PT:=ADR(buf2), SIZE:=SIZEOF(buf2), START:=0, STOP:=size2 - 1));
	ELSE
		mode := 0;
		DONE := TRUE;
	END_IF;
	pos := pos + size1;
END_CASE;

run_last := RUN;

(* revision history

ks	6. dec. 2009 rev 1.0
	original version

*)

END_FUNCTION_BLOCK

// POUs/CONVERT/BASE64_DECODE_STREAM
FUNCTION_BLOCK BASE64_DECODE_STREAM
VAR_IN_OUT
	BUF1 : ARRAY [0..63] OF BYTE;
	BUF2 : ARRAY [0..47] OF BYTE;
END_VAR
VAR_INPUT
	SIZE1 : INT;
END_VAR
VAR_OUTPUT
	SIZE2 : INT;
END_VAR
VAR_TEMP
	a: INT;
	b: WORD;
	o: INT;
	off: INT;
	i1: INT;
	i2: INT;
	c: INT;
END_VAR

(*
version 1.0	06. dec. 2009
programmer 	ks
tested by	ks

BASE64_DECODE_STREAM konvertiert einzelne Base64 kodierte Datenblöcke in normalen Datenblöcke. 

*)

IF SIZE1 <= 0 THEN SIZE2 := 0; RETURN; END_IF;
c := SIZE1 - 1;
i2 := 0;
a := 0;
b := 0;
FOR i1 := 0 TO c DO
	o := BUF1[i1];
	IF o = 61  (* = *) THEN	EXIT;
	ELSIF o > 96 (* a-z *) THEN off := 71;
	ELSIF o > 64 (* A-Z *) THEN off := 65;
	ELSIF o > 47 (* 0-9 *) THEN off := -4;
	ELSIF o = 43 (* + *) THEN off := -19;
	ELSIF o = 47 (* / *) THEN off := -16;
	END_IF;
	b := SHL(b,6) OR INT_TO_BYTE(o - off);
	a := a + 6;
	IF a >= 8 THEN
		a := a - 8;
		BUF2[i2] := WORD_TO_BYTE(SHR(b,a));
		i2 := i2 + 1;
		b := b AND NOT SHL(WORD#16#FFFF,a);
	END_IF;
END_FOR;
SIZE2 := i2;

(* revision history

ks	6. dec. 2009 rev 1.0
	original version

*)

END_FUNCTION_BLOCK

// POUs/DEMO/BASE64_DEMO
PROGRAM BASE64_DEMO
VAR
	text1: STRING(144) := '<4036.1076324381@guildenstern.zeitform.de>';
	text2: STRING(192);
	text3: STRING(144);
	BASE64_DECODE_STR: BASE64_DECODE_STR;
	BASE64_ENCODE_STR: BASE64_ENCODE_STR;
	start: BOOL := TRUE;
	done1: BOOL;
	done2: BOOL;
END_VAR

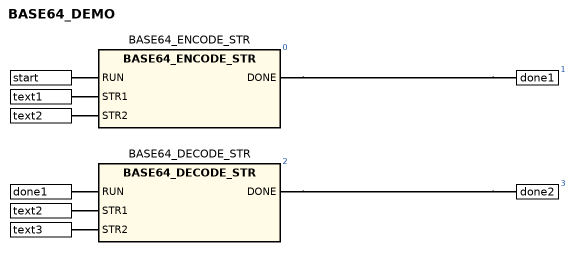
BASE64_ENCODE_STR(RUN := start, STR1 := text1, STR2 := text2);
done1 := BASE64_ENCODE_STR.DONE;
BASE64_DECODE_STR(RUN := done1, STR1 := text2, STR2 := text3);
done2 := BASE64_DECODE_STR.DONE;

END_PROGRAM

// POUs/CONVERT/BASE64_ENCODE_STR
FUNCTION_BLOCK BASE64_ENCODE_STR
VAR_INPUT
	RUN : BOOL;
END_VAR
VAR_OUTPUT
	DONE : BOOL;
END_VAR
VAR_IN_OUT
	STR1 : STRING(144);
	STR2 : STRING(192);
END_VAR
VAR
	BASE64_ENCODE_STREAM : BASE64_ENCODE_STREAM;
	run_last : BOOL;
	buf1 : ARRAY [0..47] OF BYTE;
	buf2 : ARRAY [0..63] OF BYTE;
	mode : INT;
	size1 : INT;
	size2 : INT;
	end : INT;
	pos : INT;
END_VAR

(*
version 1.0	06. dec. 2009
programmer 	ks
tested by	ks

BASE64_ENCODE_STR konvertiert einen normalen String in einen BASE64 kodierten String. 

*)

CASE mode OF
0:	IF RUN AND NOT run_last THEN
		DONE := FALSE;
		mode := 1;
		end := LEN(STR1);
		pos := 0;
		STR2 := '';
	END_IF;
1:
	size1 := MIN(48,end - pos);
	IF size1 > 0 THEN
		OSCAT_BASIC._STRING_TO_BUFFER(STR:=MID(STR1, size1, pos + 1), POS:=0, PT:=ADR(buf1), SIZE:=SIZEOF(buf1));
		BASE64_ENCODE_STREAM(BUF1:=buf1 ,BUF2:=buf2 ,SIZE1:=size1 ,SIZE2=>size2);
		STR2 := CONCAT(STR2,OSCAT_BASIC.BUFFER_TO_STRING(PT:=ADR(buf2), SIZE:=SIZEOF(buf2), START:=0, STOP:=size2 - 1));
	ELSE
		mode := 0;
		DONE := TRUE;
	END_IF;
	pos := pos + size1;
END_CASE;

run_last := RUN;

(* revision history

ks	6. dec. 2009 rev 1.0
	original version

*)

END_FUNCTION_BLOCK

// POUs/CONVERT/BASE64_ENCODE_STREAM
FUNCTION_BLOCK BASE64_ENCODE_STREAM
VAR_IN_OUT
	BUF1 : ARRAY [0..47] OF BYTE;
	BUF2 : ARRAY [0..63] OF BYTE;
END_VAR
VAR_INPUT
	SIZE1 : INT;
END_VAR
VAR_OUTPUT
	SIZE2 : INT;
END_VAR
VAR
	a: INT;
	b: WORD;
	i: INT;
	i2: INT;
	i3: INT;
	c: INT;
	BASE64: STRING(64) := 'ABCDEFGHIJKLMNOPQRSTUVWXYZabcdefghijklmnopqrstuvwxyz0123456789+/';
END_VAR

(*
version 1.0	06. dec. 2009
programmer 	ks
tested by	ks

BASE64_ENCODE_STREAM konvertiert Datenblöcke in Base64. 

*)

IF SIZE1 <= 0 THEN
	SIZE2 := 0;
	RETURN;
END_IF;
c := SIZE1 - 1;
i2 := 0;
a := 0;
b := 0;
FOR i := 0 TO c DO
	b := SHL(b,8) OR BUF1[i];
	a := a + 8;
	WHILE a >= 6 DO
		a := a - 6;
		buf2[i2] := OSCAT_BASIC.CODE(BASE64,WORD_TO_INT(SHR(b,a)) + 1);
		i2 := i2 + 1;
		b := b AND NOT SHL(WORD#16#FFFF,a);
	END_WHILE;
END_FOR;
IF a > 0 THEN
	buf2[i2] := OSCAT_BASIC.CODE(BASE64,WORD_TO_INT(SHL(b,6 - a)) + 1);
	i2 := i2 + 1;
	i3 := i2 + (NOT INT_TO_WORD(i2) AND 2#11);
	FOR i := i2 TO i3 DO
		buf2[i] := 61;
	END_FOR;
	SIZE2 := i3 + 1;
ELSE
	SIZE2 := i2;
END_IF;

(* revision history

ks	6. dec. 2009 rev 1.0
	original version

*)

END_FUNCTION_BLOCK

// POUs/FILE/CSV_PARSER_BUF
FUNCTION_BLOCK CSV_PARSER_BUF
VAR_INPUT
	SEP : BYTE;
END_VAR
VAR_IN_OUT
	RUN : BYTE;
	OFFSET : UDINT;
	VALUE : STRING(OSCAT_BASIC.STRING_LENGTH);
	PT : NETWORK_BUFFER;
END_VAR
VAR_OUTPUT
	RESULT : BYTE;
END_VAR
VAR
	step : INT;
	size : INT;
	c : BYTE;
	v_add : BYTE;
	i : INT;
	state : BYTE;
	eof : BOOL;
	pv : POINTER TO BYTE;
	pve : DWORD;
	watchdog : TON;
	x : BOOL;

	(*LOG_MSG : LOG_MSG;
	_debug_enable : BOOL := TRUE;
	step_last : INT;*)
END_VAR

(*
version 1.0		01. oct. 2010
programmer 		ks
tested by			ks

CSV_PARSER_BUF liefert die Elemente oder Zeilen einer Textdatei die in einem Bytearray abgelegt ist.

--------------------------------------

RUN Mode
00 = kein Befehl aktiv
01 = Element suchen

Result Codes
01 = Element gefunden
02 = Element und Zeilenende erkannt
05 = Befehl in Arbeit (Busy)
10 = nichts gefunden - Daten-Ende erreicht

State Codes
01 = Element gefunden
02 = Element und Zeilenende erkannt
05 = Befehl in Arbeit (Busy)
10 = nichts gefunden - Daten-Ende erreicht

*)

IF RUN > 0 THEN
	IF state = 0 THEN (* Auswertung neu beginnen *)

		pv := ADR(VALUE);
		pv^ := 0; (* VALUE = '' *)
		pve := pv + INT_TO_DWORD(OSCAT_BASIC.STRING_LENGTH);
		i := UDINT_TO_INT(OFFSET);
		size := UINT_TO_INT(PT.SIZE) - 1;
		RESULT := 0;
		state := 5; (* Befehl in Arbeit (Busy) *)
		step := 0; (* Auswertung neu beginnen *)

		(* ---------------- Debug-Message -----------------------*)
		(*IF _debug_enable THEN
			LOG_CL.NEW_MSG := 'CPF: Startindex: ~1';
			LOG_CL.PRINTF[1] := INT_TO_STRING(i);
			LOG_MSG();
		END_IF;*)
		(* -----------------------------------------------------------------*)

	END_IF;

	watchdog(IN:=FALSE,PT:=T#1ms); (* Timer neustarten *)
	watchdog.IN := TRUE;

	WHILE (state = 5) DO (* Schleife solange kein Ergebnis *)

		watchdog(); (* Timer aktualisieren *)

		IF watchdog.Q THEN (* watchdog ausgelöst *)
			state := 5;
			EXIT;
		ELSIF i > size THEN (* kein weiteres zeichen vorhanden *)
			state := 10; (* nichts gefunden - Daten-Ende erreicht *)
			EXIT;
		ELSE

			c := PT.BUFFER[i]; (* neues Zeichen aus Buffer lesen *)
			eof := i + 1 = PT.SIZE; (* End of File *)

			v_add := 0;

			IF c = SEP THEN (* Neues Element erkannt *)
				state := 1;
				x := TRUE;
			ELSIF c >= 32 THEN (* Element erkannt *)
				v_add := c; (* Zeichen ablegen *)
				IF eof THEN
					state := 2; (* Element und Zeilenende erkannt *)
				ELSE
					x := TRUE;
				END_IF;
			ELSE
				IF x THEN
					state := 2; (* Element und Zeilenende erkannt *)
					x := FALSE;
				END_IF;
			END_IF;

			IF v_add > 0  AND pv < pve THEN (* Zeichen zu Value-String hinzufügen *)
				pv^ := v_add; (* Zeichen eintragen *)
				pv := pv + 1;
				pv^ := 0; (* String-Terminierung eintragen *)
			END_IF;

			i := i + 1; (* Datenzeiger erhöhen *)

		END_IF;
	END_WHILE;

	CASE state OF
	01:	(* Element gefunden *)
		RESULT := 1; (* Element gefunden *)
		OFFSET := i; (* Offset uebernehmen *)
		RUN := 0;
		state := 0;
	02:	(* Element gefunden *)
		RESULT := 2; (* Element und Zeilenende erkannt *)
		OFFSET := i; (* Offset uebernehmen *)
		RUN := 0;
		state := 0;

	05:	RESULT := 5; (* in Arbeit *)

	10:	(* Indexüberschreitung - Bufferende *)
		RESULT := 10; (* nichts gefunden - Datenende erreicht *)
		OFFSET := i; (* Offset uebernehmen *)
		RUN := 0;
		state := 0;
	END_CASE;

	(* ---------------- Debug-Message -----------------------*)
	(*IF _debug_enable THEN
		LOG_CL.NEW_MSG := 'CPF: intern Result ~1 , state ~2, step ~3 , offset ~4, run ~5';
		LOG_CL.PRINTF[1] := BYTE_TO_STRING(RESULT);
		LOG_CL.PRINTF[2] := BYTE_TO_STRING(state);
		LOG_CL.PRINTF[3] := INT_TO_STRING(step);
		LOG_CL.PRINTF[4] := UDINT_TO_STRING(OFFSET);
		LOG_CL.PRINTF[5] := BYTE_TO_STRING(RUN);
		LOG_MSG();
	END_IF;*)
	(* -----------------------------------------------------------------*)

END_IF;

(* ---------------- Debug-Message -----------------------*)
(*IF _debug_enable THEN
	IF step_last <> step THEN
		LOG_CL.NEW_MSG := 'IPB: Step: ~1';
		LOG_CL.PRINTF[1]  := INT_TO_STRING(step);
		LOG_MSG();
	END_IF;
	step_last := step;
END_IF;*)
(* -----------------------------------------------------------------*)

(* revision history
ks	01. oct. 2010	rev 1.0
	original version
*)

END_FUNCTION_BLOCK

// POUs/OTHER/LOG_MSG
FUNCTION_BLOCK LOG_MSG
(* VAR_EXTERNAL
	LOG_CL :	LOG_CONTROL;
END_VAR *)
VAR
	FB_PRINT_SF :PRINT_SF;
	idX : INT;
END_VAR

(*
version 1.0		01 mai 2010
programmer		ks
tested by		ks

LOG_MSG trägt Meldungen in den Loggingbuffer ein
*)

IF DWORD_TO_BYTE(SHL(LOG_CL.NEW_MSG_OPTION,16)) > LOG_CL.LEVEL THEN RETURN; END_IF; (* Logging freigegeben ?*)

FB_PRINT_SF(PRINTF_DATA := LOG_CL.PRINTF,STR := LOG_CL.NEW_MSG);

IF LOG_CL.RESET THEN (* Logeinträge löschen *)
	LOG_CL.RESET := FALSE;
	LOG_CL.RING_MODE := FALSE;
	LOG_CL.IDX := 0;
	LOG_CL.UPDATE_COUNT := LOG_CL.UPDATE_COUNT + UINT#1; (* UpdateCount erhöhen *)
END_IF;

IF LOG_CL.SIZE > 0 THEN (* size wert ist eingetragen *)
	IF LEN(LOG_CL.NEW_MSG) > 0 THEN (* Meldung in Puffer eintragen *)
		IF (LOG_CL.IDX >= LOG_CL.SIZE) THEN
			LOG_CL.RING_MODE := TRUE; (* bei Überlauf = Ringbuffermodus *)
			LOG_CL.IDX := 0; (* wieder auf arrayanfang positionieren *)
		END_IF;

		LOG_CL.UPDATE_COUNT := LOG_CL.UPDATE_COUNT + UINT#1; (* UpdateCount erhöhen *)
		LOG_CL.IDX := LOG_CL.IDX + INT#1; (* nächste freie Position *)
		idx := LOG_CL.IDX; (* lade aktuelle Log-Puffer Positition *)
		LOG_CL.MSG[idx] := LOG_CL.NEW_MSG; (* neuen Log-String in puffer ablegen  *)
		LOG_CL.MSG_OPTION[idx] := LOG_CL.NEW_MSG_OPTION; (* neue Log-String Option in puffer ablegen  *)
		LOG_CL.NEW_MSG := ''; (* letzten Log-String löschen *)
	END_IF;
END_IF;

END_FUNCTION_BLOCK

// POUs/OTHER/PRINT_SF
FUNCTION_BLOCK PRINT_SF
VAR_IN_OUT
	PRINTF_DATA : PRINTF_DATA;
	STR : STRING(LOG_SIZE);
END_VAR
VAR
	pos : INT;
	c : INT;
	src : STRING(1) := '~';
	run : BOOL;
END_VAR

(*

version 1.0 		14. aug. 2009
programmer 	ks
tested by		ks

PRINTF erzeugt aus einem Parameterstring und den übergebenen Parameterdaten einen Text
*)

IF LEN(STR) > 0 THEN
	run := TRUE;

	WHILE (run) DO
		pos := FIND(STR,src);
		PRINTF_DATA[10] := '';

		IF pos = 0 THEN
			run:= FALSE;
		ELSE
			c := OSCAT_BASIC.CODE(STR:=STR,POS:=pos + 1);
			IF OSCAT_BASIC.ISC_NUM(INT_TO_BYTE(c)) THEN
				c := c - 48; (* notwendig weil innerhalb einer indexangabe nur eine var stehen darf *)
				PRINTF_DATA[10] := PRINTF_DATA[c]; (* Kommando 1-9 ergibt Parameterindex 1-9 *)
				(* Parameter gegen Text tauschen *)
			END_IF;
			IF LEN(PRINTF_DATA[10]) + LEN(STR) > LOG_SIZE THEN
				PRINTF_DATA[10] := '..';
			END_IF;
			(* pcworx: aus und eingangsstring muss verschieden sein *)
			PRINTF_DATA[11] := STR;
			STR := REPLACE(PRINTF_DATA[11],PRINTF_DATA[10],2,pos);
		END_IF;
	END_WHILE;
END_IF;

(* revision history

ks	14. aug. 2009	rev 1.0
	original version

*)

END_FUNCTION_BLOCK

// POUs/DEMO/CSV_PARSER_BUF_DEMO
PROGRAM CSV_PARSER_BUF_DEMO
VAR CONSTANT
	 line_cnt : INT:=2;
	 col_cnt : INT:=4;
END_VAR
VAR
	CPB : CSV_PARSER_BUF;
	FS : FILE_SERVER;
	FSD : FILE_SERVER_DATA;
	PT : NETWORK_BUFFER;
	sep : BYTE;
	value : STRING(OSCAT_BASIC.STRING_LENGTH);
	step : INT;
	result : BYTE;
	offset : UDINT;
	run : BYTE;
	done : BOOL;
	value_real : REAL;
	cnt : INT;
	line : INT;
	idx : INT;
	data : ARRAY [1..line_cnt, 1..col_cnt] OF REAL;

	(*LOG_MSG : LOG_MSG;
	_debug_enable : BOOL := TRUE;*)
END_VAR

(* Demo-Programm: CSV-Datei mittels Enumeration auswerten
die groesse des arrays kann mittels konstanten line_cnt und col_cnt angepasst werden

 ----- den nachfolgenden Textblock als datei "csv.txt" auf der sps ablegen ---
10.45,20,30,40.8
115,3450.2123,456,123.1
---------------------------------------------------------------------------------*)

CASE step OF

00:	IF NOT done THEN
	 	(* File_Daten einrichten  *)
		FSD.FILENAME := 'csv.txt'; (* Dateiname *)
		FSD.MODE := 1; (* vorhandene Datei zum lesen öffnen *)
		FSD.OFFSET := 0; (* Start bei Dateianfang *)
		PT.SIZE := 65535; (* maximale länge einlesen *)
		step := 10;
	END_IF;

10:	IF FSD.MODE = 0 THEN (* Datei geöffnet ? *)
		OFFSET := 0; (* Start Offset vorgeben *)
		sep :=44; (* Trennzeichen , *)
		run := 1; (* Element suchen *)
		cnt := 0;
		step := 20;
	END_IF;

20:	IF run = 0 THEN
		(* ---------------------- Debug-Message ----------------------------*)
		(*IF _debug_enable THEN
			LOG_CL.NEW_MSG := 'CPFD: /value >~2< /offset ~3 /Run ~4 /Result ~5';
			LOG_CL.PRINTF[2] := value;
			LOG_CL.PRINTF[3] := UDINT_TO_STRING(OFFSET);
			LOG_CL.PRINTF[4] := BYTE_TO_STRING(run);
			LOG_CL.PRINTF[5] := BYTE_TO_STRING(result);
			LOG_MSG();
		END_IF;*)
		(* -----------------------------------------------------------------*)

		run := 1; (*  nächstes Element suchen  *)

		IF result = 1 OR result = 2 THEN
			(* automatische konvertierung in real ausführen *)
			IF LEN(value) <= 20 THEN
				value_real := OSCAT_BASIC.FLOAT_TO_REAL(FLT:=value);
			ELSE
				value_real := 0.0;
			END_IF;

			cnt := cnt + 1;
			IF cnt <= line_cnt * col_cnt THEN
				line := (cnt / col_cnt) + 1;
				idx := (cnt MOD col_cnt);
				data[line,idx] := value_real; (* Daten in Array eintragen *)
			END_IF;

		ELSIF result = 10 THEN (* nichts mehr gefunden *)
			run := 0; (* keine weitere INI Auswertung erwünscht *)
			FSD.MODE := 5; (* Datei schliessen *)
			step := 30;
		END_IF;
	END_IF;

30:	IF FSD.MODE = 0 THEN (* Datei geschlossen ? *)
		step := 0;
		done := TRUE;
	END_IF;

END_CASE;

CPB(SEP:=sep,RUN:=run,OFFSET:=OFFSET,VALUE:=value,PT:=PT,RESULT=>result); (* CSV PARAMETER BUF *)
FS(FSD:=FSD,PT:=PT); (* FILE_SERVER *)

END_PROGRAM

// POUs/HARDWARE/FILE_SERVER
FUNCTION_BLOCK FILE_SERVER
VAR_IN_OUT
	FSD : FILE_SERVER_DATA;
	PT : NETWORK_BUFFER;
END_VAR
VAR
	buf_size : UDINT;
	handle : DWORD;
	read_max_length : UDINT;
	file_position : UDINT;
	used_filename : STRING;
	length_read : UDINT;
	write_length : UDINT;
	length_written : UDINT;
	open_handle : DWORD;
	seek_position : UDINT;
	tell_position : UDINT;
	file_size : DINT;
	open_mode : STRING(2);
	last_mode: BYTE;
	command : BYTE;
	error_code : BYTE;
	error : BOOL;
	file_change : BOOL;
	step : INT;
	FSR : FILE_SERVER_RUNTIME;

	(*step_last : INT;
	FB_LOG_MESSAGE : LOG_MSG;
	_debug_enable : BOOL := TRUE;*)
END_VAR
(*
version 1.2		08. mar. 2016
programmer 		ks
tested by			ks

FILE_SERVER ermöglicht den Zugriff auf Datteien mittels Plattform-Neutraler Schnittstelle
*)

(*
1 = File_Open_Exist + File_Read
2 = File_Open_Exist + File_Write
3 = File_Open_New   + File_Write
4 = File_Remove
5 = File_Close

- Action -
1 = file_open   (open)
2 = file_close  (close)
3 = file_read   (read)
4 = file_write  (write)
5 = file_seek   (setpos)
6 = file_tell   (getpos)
7 = file_remove (delete)

---- fehlermeldungen----

0						Kein Fehler
1	SysFileOpen		Fehler
2	SysFileClose		Fehler
3	SysFileRead		Fehler
4	SysFileWrite		Fehler
5	SysFileSetPos	Fehler
6	SysFileGetPos	Fehler
7	SysFileDelete		Fehler
8	SysFileGetSize	Fehler
255	Applikation	Position liegt hinter dem Dateiende

*)

CASE step OF
0:
	IF FSD.MODE = LIMIT(1,FSD.MODE,5) THEN

		(* ---------------------- Debug-Message ----------------------------*)
		(*IF _debug_enable THEN
			LOG_CL.NEW_MSG := 'File_Start Mode=~1';
			LOG_CL.PRINTF[1] := BYTE_TO_STRING(FSD.MODE);
			FB_LOG_MESSAGE();
		END_IF;*)
		(* -----------------------------------------------------------------*)

		buf_size := SIZEOF(PT.BUFFER);

		IF FSD.MODE = 4 THEN (* File_Remove *)
			IF handle > 0 THEN
				File_change := TRUE;
				step := 32000; (* File_Close ausführen *)
			ELSE
				step := 90; (* File_Remove ausführen *)
			END_IF;

		ELSIF FSD.MODE = 5 THEN (* File_Close *)
			step := 32000; (* File_Close ausführen *)

		ELSIF handle = 0 THEN (* MODE 1,2,3 *)
			step := 100; (* File muss erst geöffnet werden *)

		ELSE (* File ist geöffnset *)
			IF used_filename = FSD.FILENAME AND FSD.MODE = last_mode THEN (* kein Moduswechsel ? *)
				step := 200; (* ohne open prozedure weitermachen *)
			ELSE
				step := 32000;
				File_change := TRUE;
			END_IF;
		END_IF;
	END_IF;

(* ----------------------------------- *)
090: (* File_Remove *)
	command := 7; (* File Remove *)
	step := 95;

095: (* File_Remove beendet *)
	IF command = 0 THEN
		step := 30000; (* Beenden *)
	END_IF;
(* ----------------------------------- *)

100: (* File Size - Dateigroesse bestimmen *)
	command := 8; (* File Size *)
	step := 110;

110: (* File Size beendet *)
	IF command = 0 THEN
		IF FSD.MODE = 1 THEN (* open + read *)
			open_mode := 'r';
			FSD.FILE_SIZE := file_size; (* aktuelle Dateigroesse *)
		ELSIF FSD.MODE = 2 THEN (* open + write *)
			open_mode := 'a';
			FSD.FILE_SIZE := file_size; (* aktuelle Dateigroesse *)
		ELSE (* open new + write *)
			open_mode := 'w';
			FSD.FILE_SIZE := 0; (* aktuelle Dateigroesse *)
		END_IF;
		command := 1; (* File Open *)
		last_mode := FSD.MODE;
		step := 150; (* File_Open ausführen *)
	END_IF;

150: (* File Open *)
	IF command = BYTE#0 THEN
		IF error THEN
			step := 30000; (* Beenden *)
		ELSE
			(* Filedaten eintragen *)
			handle := open_handle;
			used_filename := FSD.FILENAME;
			file_position := UDINT#4294967295; (* maximal = unbekannt *)
			FSD.FILE_OPEN := TRUE;
			step := 200;
		END_IF;
	END_IF;

200: (* File Seek *)
	IF FSD.OFFSET = UDINT#4294967294 THEN (* 16#FFFF_FFFE -> Zeiger auf Dateiende stellen *)
		command := 5; (* File-Seek *)
		seek_position := FSD.FILE_SIZE;
		step := 210;
	ELSIF FSD.OFFSET > FSD.FILE_SIZE THEN (* prüfe auf gültige offset-vorgabe *)
		error_code := 255;
		step := 30000; (* Beenden *)
	ELSIF FSD.OFFSET <> file_position THEN
		command := 5; (* File-Seek *)
		seek_position := FSD.OFFSET;
		step := 210;
	ELSE
		step := 300;
	END_IF;

210: (* File Seek *)
	IF command = 0 THEN
		file_position := seek_position;
		IF error THEN
			step := 30000; (* Beenden *)
		ELSE
			step := 300;
		END_IF;
	END_IF;

300: (* Read or Write ? *)
	IF FSD.MODE = 1 THEN
		step := 400; (* Read *)
	ELSE
		step := 500; (* Write *)
	END_IF;

400: (* File Read *)
	IF UINT_TO_UDINT(PT.SIZE) > buf_size THEN (* Leselänge auf Buffergroesse begrenzen *)
		read_max_length := buf_size;
	ELSE
		read_max_length := UINT_TO_UDINT(PT.SIZE);
	END_IF;

	(* Leselänge an Dateilänge anpassen *)
	IF file_position + read_max_length > FSD.FILE_SIZE THEN
		read_max_length := FSD.FILE_SIZE - file_position;
	END_IF;

	IF read_max_length > 0 THEN
		command := 3; (* File_Read *)
		step := 410;
	ELSE
		PT.SIZE := UINT#0;
		step := 30000; (* Beenden *)
	END_IF;

410: (* File Read *)
	IF command = 0 THEN
		PT.SIZE := UDINT_TO_UINT(length_read);
		IF NOT Error THEN
			file_position := file_position + length_read; (* aktueller File_Position korrigieren *)
			FSD.OFFSET := file_position;
		END_IF;
		step := 30000; (* Beenden *)
	END_IF;

500: (* File Write *)
	IF UINT_TO_UDINT(PT.SIZE) > buf_size THEN (* Schreiblänge auf Buffergroesse begrenzen *)
		write_length := buf_size;
	ELSE
		write_length := UINT_TO_UDINT(PT.SIZE);
	END_IF;

	IF write_length > 0 THEN
		command := 4; (* File_Write *)
		step := 510;
	ELSE
		step := 30000; (* Beenden *)
	END_IF;

510:
	IF command = 0 THEN
		IF NOT Error THEN
			file_position := file_position + length_written; (* aktueller File_Position korrigieren *)
			FSD.OFFSET := file_position;
			IF file_position > FSD.FILE_SIZE THEN (* Datei ist groesser geworden *)
				FSD.FILE_SIZE := file_position;
			END_IF;
		END_IF;
		step := 30000; (* Beenden *)
	END_IF;

 (* --------------------------------------------- *)

30000: (* Befehl fertig *)
	FSD.MODE := 0;
	FSD.ERROR := error_code;
	step := 0;

	(* ---------------- Debug-Message -----------------------*)
	(*IF _debug_enable THEN
		LOG_CL.NEW_MSG := 'File_Stop: File ~1, error ~7, code ~8';
		LOG_CL.PRINTF[1]  := used_filename;
		LOG_CL.PRINTF[7]  := INT_TO_STRING(BOOL_TO_INT(error));
		LOG_CL.PRINTF[8]  := BYTE_TO_STRING(error_code);
		FB_LOG_MESSAGE();
	END_IF;*)
	(* --------------------------------------------- *)

32000:
	IF handle > 0 THEN
		command := 2; (* File_Close ausführen *)
	END_IF;
	step := 32100;

32100:
	IF command = 0 THEN (* File Close beendet *)
		(* Filedaten ablöschen *)
		FSD.FILE_OPEN := FALSE;
		file_position := 0;
		FSD.FILE_SIZE := 0;
		FSD.OFFSET := 0;
		used_filename := '';
		handle := 0;

		(* File_Name wurde fliegend geändert ? *)
		IF File_change THEN
			File_change := FALSE;
			step := 0;
		ELSE
			step := 30000;
		END_IF;
	END_IF;

END_CASE;

(* 1 = file_open
   2 = file_close
   3 = file_read
   4 = file_write
   5 = file_seek
   6 = file_tell
   7 = file_remove
*) 

FSR(MODE:=BYTE#0,COMMAND:=command,FSD:=FSD); (* File server Runtime / Befehlsstart überwachen *)

(* ------------ File Open ------------- *)
IF command = 1 THEN
	open_handle := SysFileOpen(FSD.FILENAME,open_mode);
	error := open_handle = 0;
	error_code := SEL(error,0,command);
	command := 0;
	FSR(MODE:=BYTE#1,COMMAND:=command,FSD:=FSD); (* File server Runtime / Befehlstop überwachen *)
	(* ---------------- Debug-Message -----------------------*)
	(*IF _debug_enable THEN
		LOG_CL.NEW_MSG := 'Open: File ~1, handle ~2 , mode ~3 , error ~7, code ~8';
		LOG_CL.PRINTF[1] := FSD.FILENAME;
		LOG_CL.PRINTF[2] := DWORD_TO_STRING(open_handle);
		LOG_CL.PRINTF[3] := open_mode;
		LOG_CL.PRINTF[7] := INT_TO_STRING(BOOL_TO_INT(error));
		LOG_CL.PRINTF[8] := BYTE_TO_STRING(error_code);
		FB_LOG_MESSAGE();
	END_IF;*)
	(* -----------------------------------------------------------------*)
END_IF;

(* ----------- File Close ------------- *)
IF command = 2 THEN
	error := NOT SysFileClose(handle);
	error_code := SEL(error,0,command);
	command := 0;
	FSR(MODE:=BYTE#1,COMMAND:=command,FSD:=FSD); (* File server Runtime / Befehlstop überwachen *)
	(* ---------------- Debug-Message -----------------------*)
	(*IF _debug_enable THEN
		LOG_CL.NEW_MSG := 'Close: File ~1, error ~7, code ~8';
		LOG_CL.PRINTF[1] := used_filename;
		LOG_CL.PRINTF[7] := INT_TO_STRING(BOOL_TO_INT(error));
		LOG_CL.PRINTF[8] := BYTE_TO_STRING(error_code);
		FB_LOG_MESSAGE();
	END_IF;*)
	(* -----------------------------------------------------------------*)
END_IF;

(* ------------ File Read ------------- *)
IF command = 3 THEN
	length_read := SysFileRead(handle, ADR(PT.BUFFER), read_max_length);
	error := length_read = 0;
	error_code := SEL(error,0,command);
	command := 0;
	FSR(MODE:=BYTE#1,COMMAND:=command,FSD:=FSD); (* File server Runtime / Befehlstop überwachen *)
	(* ---------------- Debug-Message -----------------------*)
	(*IF _debug_enable THEN
		LOG_CL.NEW_MSG := 'Read: File ~1, soll ~2,ist ~3 ,error ~7, code ~8';
		LOG_CL.PRINTF[1] := used_filename;
		LOG_CL.PRINTF[2] := UDINT_TO_STRING(read_max_length);
		LOG_CL.PRINTF[3] := UDINT_TO_STRING(length_read);
		LOG_CL.PRINTF[7] := INT_TO_STRING(BOOL_TO_INT(error));
		LOG_CL.PRINTF[8] := BYTE_TO_STRING(error_code);
		FB_LOG_MESSAGE();
	END_IF;*)
	(* -----------------------------------------------------------------*)
END_IF;

(* ------------ File Write ------------- *)
IF command = 4 THEN
	length_written := SysFileWrite(handle, ADR(PT.BUFFER), write_length);
	error := length_written = 0;
	error_code := SEL(error,0,command);
	command := 0;
	FSR(MODE:=BYTE#1,COMMAND:=command,FSD:=FSD); (* File server Runtime / Befehlstop überwachen *)
	(* ---------------- Debug-Message -----------------------*)
	(*IF _debug_enable THEN
		LOG_CL.NEW_MSG := 'Write: File ~1, soll ~2,ist ~3 ,error ~7, code ~8';
		LOG_CL.PRINTF[1] := used_filename;
		LOG_CL.PRINTF[2] := UDINT_TO_STRING(write_length);
		LOG_CL.PRINTF[3] := UDINT_TO_STRING(length_written);
		LOG_CL.PRINTF[7] := INT_TO_STRING(BOOL_TO_INT(error));
		LOG_CL.PRINTF[8] := BYTE_TO_STRING(error_code);
		FB_LOG_MESSAGE();
	END_IF;*)
	(* -----------------------------------------------------------------*)
END_IF;

(* ------------ File Seek ------------- *)
IF command = 5 THEN
	error := NOT SysFileSetPos(handle, seek_position);
	error_code := SEL(error,0,command);
	command := 0;
	FSR(MODE:=BYTE#1,COMMAND:=command,FSD:=FSD); (* File server Runtime / Befehlstop überwachen *)
	(* ---------------- Debug-Message -----------------------*)
	(*IF _debug_enable THEN
		LOG_CL.NEW_MSG := 'Seek: File ~1,pos ~3 ,error ~7, code ~8';
		LOG_CL.PRINTF[1] := used_filename;
		LOG_CL.PRINTF[3] := UDINT_TO_STRING(seek_position);
		LOG_CL.PRINTF[7] := INT_TO_STRING(BOOL_TO_INT(error));
		LOG_CL.PRINTF[8] := BYTE_TO_STRING(error_code);
		FB_LOG_MESSAGE();
	END_IF;*)
	(* -----------------------------------------------------------------*)
END_IF;

(* ------------ File Tell ------------- *)
IF command = 6 THEN
	tell_position := SysFileGetPos(handle);
	error := tell_position < 0;
	error_code := SEL(error,0,command);
	command := 0;
	FSR(MODE:=BYTE#1,COMMAND:=command,FSD:=FSD); (* File server Runtime / Befehlstop überwachen *)
	(* ---------------- Debug-Message -----------------------*)
	(*IF _debug_enable THEN
		LOG_CL.NEW_MSG := 'Tell: File ~1, pos ~3 ,error ~7, code ~8';
		LOG_CL.PRINTF[1] := used_filename;
		LOG_CL.PRINTF[3] := UDINT_TO_STRING(tell_position);
		LOG_CL.PRINTF[7] := INT_TO_STRING(BOOL_TO_INT(error));
		LOG_CL.PRINTF[8] := BYTE_TO_STRING(error_code);
		FB_LOG_MESSAGE();
	END_IF;*)
	(* -----------------------------------------------------------------*)
END_IF;

(* ------------ File Remove ------------- *)
IF command = 7 THEN
	error := NOT SysFileDelete(FSD.FILENAME);
	error_code := SEL(error,0,command);
	command := 0;
	FSR(MODE:=BYTE#1,COMMAND:=command,FSD:=FSD); (* File server Runtime / Befehlstop überwachen *)
	(* ---------------- Debug-Message -----------------------*)
	(*IF _debug_enable THEN
		LOG_CL.NEW_MSG := 'Remove: File ~1, error ~7, code ~8';
		LOG_CL.PRINTF[1] := FSD.FILENAME;
		LOG_CL.PRINTF[7] := INT_TO_STRING(BOOL_TO_INT(error));
		LOG_CL.PRINTF[8] := BYTE_TO_STRING(error_code);
		FB_LOG_MESSAGE();
	END_IF;*)
	(* -----------------------------------------------------------------*)
END_IF;

(* ------------ File Size ------------- *)
IF command = 8 THEN
	file_size := SysFileGetSize(FSD.FILENAME);
	error_code := 0; (* kein Errorcode vorhanden *)
	command := 0;
	FSR(MODE:=BYTE#1,COMMAND:=command,FSD:=FSD); (* File server Runtime / Befehlstop überwachen *)
	(* ---------------- Debug-Message -----------------------*)
	(*IF _debug_enable THEN
		LOG_CL.NEW_MSG := 'Size: File ~1, size ~3, error ~7, code ~8';
		LOG_CL.PRINTF[1] := FSD.FILENAME;
		LOG_CL.PRINTF[3] := DINT_TO_STRING(file_size);
		LOG_CL.PRINTF[7] := INT_TO_STRING(BOOL_TO_INT(error));
		LOG_CL.PRINTF[8] := BYTE_TO_STRING(error_code);
		FB_LOG_MESSAGE();
	END_IF;*)
	(* -----------------------------------------------------------------*)
END_IF;

(* ---------------- Debug-Message -----------------------*)
(*IF _debug_enable THEN
	IF step_last <> step THEN
		LOG_CL.NEW_MSG := 'Step: ~1';
		LOG_CL.PRINTF[1] := INT_TO_STRING(step);
		FB_LOG_MESSAGE();
	END_IF;
	step_last := step;
END_IF;*)
(* -----------------------------------------------------------------*)

(* revision history
ks	08. mar. 2016	rev 1.2
	Filesystem Laufzeitmessungen

ks	02. oct. 2014	rev 1.1.1
	PCWORX SRT File Delete error

ks	05. mai. 2012	rev 1.1
	auto_close funktion entfernt

ks	23. sep. 2010	rev 1.0
	original version
*)

END_FUNCTION_BLOCK

// POUs/HARDWARE/FILE_SERVER_RUNTIME
FUNCTION_BLOCK FILE_SERVER_RUNTIME
VAR_INPUT
	MODE : BYTE;
	COMMAND : BYTE;
END_VAR
VAR_IN_OUT
	FSD : FILE_SERVER_DATA;
END_VAR
VAR
	last_command : BYTE;
	init : BOOL;
	start_tx : DWORD;
	stop_tx : DWORD;
	runtime : DWORD;
END_VAR

(*
version 1.0		08.mar. 2016
programmer 		ks
tested by			ks

FILE_SERVER_RUNTIME misst die Laufzeit der Filesystem aufrufe (min,max,cur)
*)

IF init = FALSE THEN
	init := TRUE;
	FSD.RUNTIME.TIME_FILE_OPEN_MIN := UDINT#99999999;
	FSD.RUNTIME.TIME_FILE_CLOSE_MIN := UDINT#99999999;
	FSD.RUNTIME.TIME_FILE_READ_MIN := UDINT#99999999;
	FSD.RUNTIME.TIME_FILE_WRITE_MIN := UDINT#99999999;
	FSD.RUNTIME.TIME_FILE_TELL_MIN := UDINT#99999999;
	FSD.RUNTIME.TIME_FILE_SEEK_MIN := UDINT#99999999;
	FSD.RUNTIME.TIME_FILE_DELETE_MIN := UDINT#99999999;
END_IF;

(* warten auf File_Server Befehl *)
IF MODE = BYTE#0 THEN

	(* neuen befehl erkannt *)
	IF last_command = BYTE#0 AND COMMAND <> BYTE#0 THEN

		(* read system time *)
		start_tx := OSCAT_BASIC.T_PLC_MS();

	END_IF;
END_IF;


IF MODE = BYTE#1 THEN

	(* read system time *)
	stop_tx:=  OSCAT_BASIC.T_PLC_MS();

	runtime:= (stop_tx - start_tx);

	CASE BYTE_TO_INT(COMMAND) OF

	1:	FSD.RUNTIME.TIME_FILE_OPEN_CUR := runtime; 			(* aktuelle laufzeit *)
		IF FSD.RUNTIME.TIME_FILE_OPEN_MAX < runtime THEN
			FSD.RUNTIME.TIME_FILE_OPEN_MAX := runtime;		(* neue max laufzeit *)
		END_IF;
		IF FSD.RUNTIME.TIME_FILE_OPEN_MIN > runtime THEN
			FSD.RUNTIME.TIME_FILE_OPEN_MIN := runtime;		(* neue min laufzeit *)
		END_IF;

	2:	FSD.RUNTIME.TIME_FILE_CLOSE_CUR := runtime; 			(* aktuelle laufzeit *)
		IF FSD.RUNTIME.TIME_FILE_CLOSE_MAX < runtime THEN
			FSD.RUNTIME.TIME_FILE_CLOSE_MAX := runtime;		(* neue max laufzeit *)
		END_IF;
		IF FSD.RUNTIME.TIME_FILE_CLOSE_MIN > runtime THEN
			FSD.RUNTIME.TIME_FILE_CLOSE_MIN := runtime;		(* neue min laufzeit *)
		END_IF;

	3:	FSD.RUNTIME.TIME_FILE_READ_CUR := runtime; 			(* aktuelle laufzeit *)
		IF FSD.RUNTIME.TIME_FILE_READ_MAX < runtime THEN
			FSD.RUNTIME.TIME_FILE_READ_MAX := runtime;		(* neue max laufzeit *)
		END_IF;
		IF FSD.RUNTIME.TIME_FILE_READ_MIN > runtime THEN
			FSD.RUNTIME.TIME_FILE_READ_MIN := runtime;		(* neue min laufzeit *)
		END_IF;

	4:	FSD.RUNTIME.TIME_FILE_WRITE_CUR := runtime; 			(* aktuelle laufzeit *)
		IF FSD.RUNTIME.TIME_FILE_WRITE_MAX < runtime THEN
			FSD.RUNTIME.TIME_FILE_WRITE_MAX := runtime;		(* neue max laufzeit *)
		END_IF;
		IF FSD.RUNTIME.TIME_FILE_WRITE_MIN > runtime THEN
			FSD.RUNTIME.TIME_FILE_WRITE_MIN := runtime;		(* neue min laufzeit *)
		END_IF;

	5:	FSD.RUNTIME.TIME_FILE_SEEK_CUR := runtime; 			(* aktuelle laufzeit *)
		IF FSD.RUNTIME.TIME_FILE_SEEK_MAX < runtime THEN
			FSD.RUNTIME.TIME_FILE_SEEK_MAX := runtime;		(* neue max laufzeit *)
		END_IF;
		IF FSD.RUNTIME.TIME_FILE_SEEK_MIN > runtime THEN
			FSD.RUNTIME.TIME_FILE_SEEK_MIN := runtime;		(* neue min laufzeit *)
		END_IF;

	6:	FSD.RUNTIME.TIME_FILE_TELL_CUR := runtime; 			(* aktuelle laufzeit *)
		IF FSD.RUNTIME.TIME_FILE_TELL_MAX < runtime THEN
			FSD.RUNTIME.TIME_FILE_TELL_MAX := runtime;		(* neue max laufzeit *)
		END_IF;
		IF FSD.RUNTIME.TIME_FILE_TELL_MIN > runtime THEN
			FSD.RUNTIME.TIME_FILE_TELL_MIN := runtime;		(* neue min laufzeit *)
		END_IF;

	7:	FSD.RUNTIME.TIME_FILE_DELETE_CUR := runtime; 			(* aktuelle laufzeit *)
		IF FSD.RUNTIME.TIME_FILE_DELETE_MAX < runtime THEN
			FSD.RUNTIME.TIME_FILE_DELETE_MAX := runtime;		(* neue max laufzeit *)
		END_IF;
		IF FSD.RUNTIME.TIME_FILE_DELETE_MIN > runtime THEN
			FSD.RUNTIME.TIME_FILE_DELETE_MIN := runtime;		(* neue min laufzeit *)
		END_IF;

	END_CASE;

END_IF;

last_command := COMMAND;

(* revision history

ks	08. mar. 2016	rev 1.0
	original version
*)

END_FUNCTION_BLOCK

// POUs/FILE/CSV_PARSER_FILE
FUNCTION_BLOCK CSV_PARSER_FILE
VAR_INPUT
	SEP : BYTE;
END_VAR
VAR_IN_OUT
	FILENAME : STRING;
	FSD : FILE_SERVER_DATA;
	RUN : BYTE;
	OFFSET : UDINT;
	VALUE : STRING(OSCAT_BASIC.STRING_LENGTH);
	PT	: NETWORK_BUFFER;
END_VAR
VAR_OUTPUT
	RESULT : BYTE;
END_VAR
VAR
	i : UDINT;
	state : BYTE;
	e : BYTE;
	mode : BYTE;
	step : INT;
	c : BYTE;
	v_add : BYTE;
	eof : BOOL;
	pv : POINTER TO BYTE;
	pve : DWORD;
	watchdog : TON;
	x : BOOL;
	FB : FILE_BLOCK;

	(*LOG_MSG : LOG_MSG;
	_debug_enable : BOOL := FALSE;
	step_last : INT;*)
END_VAR

(*
version 1.0		01. oct. 2010
programmer 		ks
tested by			ks

CSV_PARSER_FILE liefert die Elemente oder Zeilen einer Textdatei.

--------------------------------------

RUN Mode
00 = kein Befehl aktiv
01 = Element suchen

Result Codes
01 = Element gefunden
02 = Element und Zeilenende erkannt
05 = Befehl in Arbeit (Busy)
10 = nichts gefunden - Daten-Ende erreicht

State Codes
01 = Element gefunden
02 = Element und Zeilenende erkannt
05 = Befehl in Arbeit (Busy)
10 = nichts gefunden - Daten-Ende erreicht

*)

IF RUN > 0 THEN

	IF state = 0 THEN (* Auswertung neu beginnen *)
		pv := ADR(VALUE);
		pv^ := 0; (* VALUE = '' *)
		pve := pv + INT_TO_DWORD(OSCAT_BASIC.STRING_LENGTH);
		i := OFFSET;
		RESULT := 0;
		state := 5; (* Befehl in Arbeit (Busy) *)
		step := 0; (* Auswertung neu beginnen *)

		(* ---------------- Debug-Message -----------------------*)
		(*IF _debug_enable THEN
			LOG_CL.NEW_MSG := 'CPF: Startindex: ~1';
			LOG_CL.PRINTF[1] := UDINT_TO_STRING(i);
			LOG_MSG();
		END_IF;*)
		(* -----------------------------------------------------------------*)

	END_IF;

	watchdog(IN:=FALSE,PT:=T#1ms); (* Timer neustarten *)
	watchdog.IN := TRUE;

	WHILE (state = 5) DO (* Schleife solange kein Ergebnis *)

		mode := 1;
		FB(MODE:=mode,FSD:=fsd,PT:=PT,FILENAME:=FILENAME,POS:=i );
		e:=FB.ERROR;
		c:=FB.DATA;

		eof := i + 1 = FSD.FILE_SIZE; (* End of File *)

		(* ---------------- Debug-Message -----------------------*)
		(*IF _debug_enable THEN
			LOG_CL.NEW_MSG := 'CPF: mode: ~1, error: ~2 , >~7<>~3< ~4 step ~5 index ~6';
			LOG_CL.PRINTF[1] := BYTE_TO_STRING(mode);
			LOG_CL.PRINTF[2] := BYTE_TO_STRING(e);
			LOG_CL.PRINTF[3] := BYTE_TO_STRING(c);
			LOG_CL.PRINTF[4] := BOOL_TO_STRING(eof);
			LOG_CL.PRINTF[5] := INT_TO_STRING(step);
			LOG_CL.PRINTF[6] := UDINT_TO_STRING(i);
			LOG_CL.PRINTF[7] := CHR_TO_STRING(c);
			LOG_MSG();
		END_IF;*)
		(* -----------------------------------------------------------------*)
		watchdog(); (* Timer aktualisieren *)

		IF mode > 0 OR watchdog.Q THEN (* Baustein noch aktiv, oder watchdog ausgelöst *)
			state := 5;
			EXIT;
		ELSIF e > 0 THEN (* File_error oder kein weiteres zeichen vorhanden *)
			state := 10; (* nichts gefunden - Daten-Ende erreicht *)
			EXIT;
		ELSE

			v_add := 0;

			IF c = SEP THEN (* Neues Element erkannt *)
				state := 1;
				x := TRUE;
			ELSIF c >= 32 THEN (* Element erkannt *)
				v_add := c; (* Zeichen ablegen *)
				IF eof THEN
					state := 2; (* Element und Zeilenende erkannt *)
				ELSE
					x := TRUE;
				END_IF;
			ELSE
				IF x THEN
					state := 2; (* Element und Zeilenende erkannt *)
					x := FALSE;
				END_IF;
			END_IF;

			IF v_add > 0  AND pv < pve THEN (* Zeichen zu Value-String hinzufügen *)
				pv^ := v_add; (* Zeichen eintragen *)
				pv := pv + 1;
				pv^ := 0; (* String-Terminierung eintragen *)
			END_IF;

			i := i + 1; (* Datenzeiger erhöhen *)

		END_IF;
	END_WHILE;

	CASE state OF
	01:	(* Element gefunden *)
		RESULT := 1; (* Element gefunden *)
		OFFSET := i; (* Offset uebernehmen *)
		RUN := 0;
		state := 0;
	02:	(* Element gefunden *)
		RESULT := 2; (* Element und Zeilenende erkannt *)
		OFFSET := i; (* Offset uebernehmen *)
		RUN := 0;
		state := 0;

	05:	RESULT := 5; (* in Arbeit *)

	10:	(* Indexüberschreitung - Bufferende *)
		RESULT := 10; (* nichts gefunden - Datenende erreicht *)
		OFFSET := i; (* Offset uebernehmen *)
		RUN := 0;
		state := 0;
	END_CASE;

	(* ---------------- Debug-Message -----------------------*)
	(*IF _debug_enable THEN
		LOG_CL.NEW_MSG := 'CPF: intern Result ~1 , state ~2, step ~3 , offset ~4, run ~5';
		LOG_CL.PRINTF[1] := BYTE_TO_STRING(RESULT);
		LOG_CL.PRINTF[2] := BYTE_TO_STRING(state);
		LOG_CL.PRINTF[3] := INT_TO_STRING(step);
		LOG_CL.PRINTF[4] := UDINT_TO_STRING(OFFSET);
		LOG_CL.PRINTF[5] := BYTE_TO_STRING(RUN);
		LOG_MSG();
	END_IF;*)
	(* -----------------------------------------------------------------*)

END_IF;

(* ---------------- Debug-Message -----------------------*)
(*IF _debug_enable THEN
	IF step_last <> step THEN
		LOG_CL.NEW_MSG := 'CPF: Step: ~1';
		LOG_CL.PRINTF[1]  := INT_TO_STRING(step);
		LOG_MSG();
	END_IF;
	step_last := step;
END_IF;*)
(* -----------------------------------------------------------------*)

(* revision history
ks	01. oct. 2010	rev 1.0
	original version
*)

END_FUNCTION_BLOCK

// POUs/FILE/FILE_BLOCK
FUNCTION_BLOCK FILE_BLOCK
VAR_IN_OUT
	MODE : BYTE;
	FILENAME : STRING;
	FSD : FILE_SERVER_DATA;
	PT : NETWORK_BUFFER;
END_VAR
VAR_INPUT
	POS : UDINT;
END_VAR
VAR_OUTPUT
	ERROR : BYTE;
	DATA : BYTE;
END_VAR
VAR
	step : INT;
	i : INT;
	data_start : UDINT;
	data_stop : UDINT;

	(*LOG_MSG : LOG_MSG;
	_debug_enable : BOOL := TRUE;*)
END_VAR

(*
version 1.0		23. sep. 2010
programmer 		ks
tested by			ks

FILE_BLOCK liefert das angeforderte BYTE einer Datei durch einlesen von möglichst grossen Datenblöcken
*)

CASE step OF
0:	IF MODE > 0 THEN
		ERROR := 0;
		IF FSD.FILE_OPEN AND (FSD.FILE_SIZE = 0 OR POS >= FSD.FILE_SIZE) THEN
			ERROR := 255;
			MODE := 0;
		ELSIF POS < data_start OR POS > data_stop OR NOT FSD.FILE_OPEN THEN (* Daten lesen notwendig *)
			FSD.FILENAME := FILENAME;
			FSD.MODE := 1; (* open + read *)
			FSD.OFFSET := POS;
			PT.SIZE := 65535; (* maximale anzahl lesen *);
			data_start := 0;
			data_stop := 0;
			step := 10;
		ELSE (* Daten sind im Buffer vorhanden *)
			i := UDINT_TO_INT(POS - data_start); (* index berechnen *)
			DATA := PT.BUFFER[i];
			MODE := 0;
			(* ---------------------- Debug-Message ----------------------------*)
			(*IF _debug_enable THEN
				LOG_CL.NEW_MSG := 'FB: Pos: ~1 Byte: ~2 >~3<';
				LOG_CL.PRINTF[1] := UDINT_TO_STRING(POS);
				LOG_CL.PRINTF[2] := BYTE_TO_STRING(DATA);
				LOG_CL.PRINTF[3] := CHR_TO_STRING(DATA);
				LOG_MSG();
			END_IF;*)
			(* -----------------------------------------------------------------*)
		END_IF;
	END_IF;

10:	IF FSD.MODE = 0 THEN (* Befehl beendet *)
		IF FSD.ERROR > 0 THEN
			ERROR := FSD.ERROR; (* Fehler ausgeben *)
			MODE := 0;
		ELSE
			data_start := POS;
			data_stop := POS + UINT_TO_UDINT(PT.SIZE) - 1;
		END_IF;
		step := 0;
	END_IF;
END_CASE;

(* revision history
ks	23. sep. 2010	rev 1.0
	original version
*)

END_FUNCTION_BLOCK

// POUs/DEMO/CSV_PARSER_FILE_DEMO
PROGRAM CSV_PARSER_FILE_DEMO
VAR CONSTANT
	 line_cnt : INT:=2;
	 col_cnt : INT:=4;
END_VAR
VAR
	CPF : CSV_PARSER_FILE;
	FS : FILE_SERVER;
	FSD : FILE_SERVER_DATA;
	PT : NETWORK_BUFFER;
	filename : STRING;
	value :	STRING(OSCAT_BASIC.STRING_LENGTH);
	sep : BYTE;
	step : INT;
	result : BYTE;
	offset : UDINT;
	run : BYTE;
	done : BOOL;
	value_real : REAL;
	cnt : INT;
	line : INT;
	idx : INT;
	data : ARRAY [1..line_cnt, 1..col_cnt] OF REAL;

	(*LOG_MSG : LOG_MSG;
	_debug_enable : BOOL := TRUE;*)
END_VAR

(* Demo-Programm: CSV-Datei mittels Enumeration auswerten

die groesse des arrays kann mittels konstanten line_cnt und col_cnt angepasst werden

 ----- den nachfolgenden Textblock als datei "csv.txt" auf der sps ablegen ---
10.45,20,30,40.8
115,3450.2123,456,123.1
---------------------------------------------------------------------------------*)

CASE step OF

00:	IF NOT done THEN
		filename := 'csv.txt'; (* File_Daten einrichten *)
		OFFSET := 0; (* Start Offset vorgeben *)
		sep :=44; (* Trennzeichen , *)
		run := 1; (* Element suchen *)
		cnt := 0;
		step := 20;
	END_IF;

20:	IF run = 0 THEN (* kein Befehl mehr aktiv ? *)
		(* ---------------------- Debug-Message ----------------------------*)
		(*IF _debug_enable THEN
			LOG_CL.NEW_MSG := 'CPFD: /value >~2< /offset ~3 /Run ~4 /Result ~5';
			LOG_CL.PRINTF[2] := value;
			LOG_CL.PRINTF[3] := UDINT_TO_STRING(OFFSET);
			LOG_CL.PRINTF[4] := BYTE_TO_STRING(run);
			LOG_CL.PRINTF[5] := BYTE_TO_STRING(result);
			LOG_MSG();
		END_IF;*)
		(* -----------------------------------------------------------------*)

		run := 1; (*  nächstes Element suchen  *)

		IF result = 1 OR result = 2 THEN
			(* automatische konvertierung in real ausführen *)
			IF LEN(value) <= 20 THEN
				value_real := OSCAT_BASIC.FLOAT_TO_REAL(FLT:=value);
			ELSE
				value_real := 0.0;
			END_IF;

			cnt := cnt + 1;
			IF cnt <= line_cnt * col_cnt THEN
				line := (cnt / col_cnt) + 1;
				idx := (cnt MOD col_cnt);
				data[line,idx] := value_real; (* Daten in Array eintragen *)
			END_IF;

		ELSIF result = 10 THEN (* nichts mehr gefunden *)
			run := 0; (* keine weitere INI Auswertung erwünscht *)
			FSD.MODE := 5; (* Datei schliessen *)
			step := 30;
		END_IF;
	END_IF;

30:	IF FSD.MODE = 0 THEN (* Befehl Datei schliessen beendet *)
		step := 0;
		done := TRUE;
	END_IF;

END_CASE;

CPF(SEP:=sep,FILENAME:=FILENAME,FSD:=FSD,RUN:=run,OFFSET:=OFFSET,VALUE:=value,PT:=PT,RESULT=>result); (* CSV PARAMETER FILE *)
FS(FSD:=FSD,PT:=PT); (* FILE_SERVER *)

END_PROGRAM

// POUs/DATA_LOG/DLOG_BOOL
FUNCTION_BLOCK DLOG_BOOL
VAR_IN_OUT
	X : DLOG_DATA;
END_VAR
VAR_INPUT
	STATE : BOOL;
	OFF : STRING;
	ON : STRING;
	COLUMN : STRING(40);
	DELTA : BOOL;
END_VAR
VAR_OUTPUT
END_VAR
VAR
	UCB : UNI_CIRCULAR_BUFFER;
	id : WORD;
	last_delta : BOOL;
	state_last: BOOL;
END_VAR

(*
version 1.2		19. apr. 2012
programmer		ks
tested by			ks

DLOG_BOOL legt den ON/OFF Text im FIFO-RING-Buffer ab um diesen mit den Baustein DLOG_STORE_*  aufzuzeichnen
*)

CASE x.ADD_COM OF

01:	(* ADD INFO *)
	X.ID_MAX := X.ID_MAX + USINT#1;
	id := WORD#16#0601; (* Quelltype BOOL , Zieltype STRING *)
02:	(* ADD HEADER *)
	X.UCB.D_STRING := COLUMN;
	X.UCB.D_HEAD := id;
	X.UCB.D_MODE := 1;
	UCB(DATA:=X.UCB); (* Daten eintragen *)
03:	(* ADD DATA *)
	IF X.STORE_TYPE = BYTE#05 THEN (* MySQL-Modus *)
		X.UCB.D_STRING := SEL(state_last,'0','1');
	ELSE
		X.UCB.D_STRING := SEL(state_last,OFF,ON);
	END_IF;
	X.UCB.D_HEAD := id;

	X.UCB.D_MODE := 1;
	UCB(DATA:=X.UCB); (* Daten eintragen *)
	last_delta := STATE;
04:	(* ADD DATA REQ *)
	IF DELTA AND (STATE XOR last_delta) THEN
		X.ADD_DATA_REQ := TRUE;
		last_delta := STATE;
	END_IF;
END_CASE;
state_last := STATE;

(* revision history
ks	17. may. 2011	rev 1.0
	original version

ks	25. july.   2011	rev 1.1
	neue head information

ks	19. apr.   2012	rev 1.2
	code neu überarbeitet

*)

END_FUNCTION_BLOCK

// POUs/OTHER/UNI_CIRCULAR_BUFFER
FUNCTION_BLOCK UNI_CIRCULAR_BUFFER
VAR_IN_OUT
	DATA : UNI_CIRCULAR_BUFFER_DATA;
END_VAR
VAR_TEMP
	tmp_dw : DWORD;
	pTmp : POINTER TO BYTE;
	n : INT;
	n1 : INT;
	n2 : INT;
	x: BYTE;
	buf_totalsize : UINT;
END_VAR
VAR CONSTANT
	HeaderSize : INT := 4;
END_VAR
VAR
	cnt : UINT;
	mode_last : INT;

	(*LOG_MSG : LOG_MSG;
	_debug_enable : BOOL := FALSE;*)
END_VAR

(*
version 1.3		21. mar. 2016
programmer		ks
tested by			ks

UNI_CIRCULAR_BUFFER ist ein FIFO-RING-Buffer der verschiedene Datenelemente als Byte-Array aufnehmen kann.
*)

CASE DATA.D_MODE OF

01:	x := WORD_TO_BYTE(DATA.D_HEAD); (* nur rechtes byte auswerten *)
	CASE x OF
	01:	cnt := LEN(DATA.D_STRING); (* String verarbeiten *)
		pTmp := ADR(DATA.D_STRING);
	02:	cnt := 4; (* Real verarbeiten *)
		pTmp := ADR(DATA.D_REAL);
	03:	cnt := 4; (* DWORD verarbeiten *)
		pTmp := ADR(DATA.D_DWORD);
	ELSE
		cnt := 0;
	END_CASE;

	DATA.BUF_DATA_CNT := DATA.BUF_DATA_CNT + UDINT#1;

	(* ------ Daten in buffer eintragen ------ *)
	buf_totalsize := SIZEOF(DATA.BUF);

	IF (cnt + HeaderSize) > (buf_totalsize - DATA.BUF_SIZE) THEN (* genug Speicher frei ? *)
		DATA.BUF_DATA_LOST := DATA.BUF_DATA_LOST + UDINT#1;
		RETURN;
	END_IF;

	DATA.D_SIZE := cnt;

	mode_last := DATA.D_MODE;
	tmp_dw := SHL(WORD_TO_DWORD(DATA.D_HEAD),16) OR UINT_TO_DWORD(cnt);

	(* Header in Buffer eintragen *)
	n1 := 0;
	REPEAT
		n2 := MIN(HeaderSize - n1, buf_totalsize - DATA._Last);
		FOR n := 1 TO n2 DO
			tmp_dw := ROL(tmp_dw,8);
			data.BUF[DATA._Last] := DWORD_TO_BYTE(tmp_dw);
			DATA._Last := DATA._Last + 1;
		END_FOR;
		IF DATA._Last >= buf_totalsize THEN
			DATA._Last := 0;
		END_IF
		n1 := n1 + n2;
	UNTIL n1 >= HeaderSize
	END_REPEAT;

	(* Daten in Buffer eintragen *)
	n1 := 0;
	REPEAT
		n2 := MIN(cnt - n1, buf_totalsize - DATA._Last);
		FOR n := 1 TO n2 DO
			data.BUF[DATA._Last] := pTmp^;
			pTmp := pTmp + 1;
			DATA._Last := DATA._Last + 1;
		END_FOR;
		IF DATA._Last >= buf_totalsize THEN
			DATA._Last := 0;
		END_IF
		n1 := n1 + n2;
	UNTIL n1 >= cnt
	END_REPEAT;

	DATA.BUF_SIZE := DATA.BUF_SIZE + cnt + HeaderSize;
	DATA.BUF_COUNT := DATA.BUF_COUNT + 1;
	DATA.BUF_USED := UINT_TO_USINT(100 * DATA.BUF_SIZE / buf_totalsize); (* benützer Speicher in % *)
	DATA.D_MODE := 0;

	(*####################  DEBUG-MESSAGE  ###################################*)
	(*IF _debug_enable THEN
		LOG_CL.NEW_MSG := 'RP: ADD /HEAD ~1 / SIZE ~2 / CNT ~3 / >~4<';
		LOG_CL.PRINTF[1] := DWORD_TO_STRH(DATA.D_HEAD);
		LOG_CL.PRINTF[2] := UINT_TO_STRING(cnt);
		LOG_CL.PRINTF[3] := UINT_TO_STRING(DATA.BUF_COUNT);
		CASE x OF
		01:	LOG_CL.PRINTF[4] := DATA.D_STRING;
		02:	LOG_CL.PRINTF[4] := REAL_TO_STRING(DATA.D_REAL);
		03:	LOG_CL.PRINTF[4] := DWORD_TO_STRH(DATA.D_DWORD);
		ELSE
			LOG_CL.PRINTF[4] := '';
		END_CASE;
		LOG_MSG();
	END_IF;*)
	(*########################################################################*)

10..12:	(* ------ Daten aus buffer auslesen und optional löschen ------ *)
		(* 10 = nur lesen / 11 = löschen nach lesen / 12 = lesen und löschen *)
	IF DATA.D_MODE <> 11 THEN
		IF DATA.BUF_COUNT = 0 THEN RETURN; END_IF;
		buf_totalsize := SIZEOF(DATA.BUF);
		DATA._GetEnd := DATA._First;(* index des ältesten eintrags merken *)
		mode_last := DATA.D_MODE;
	
		(* Header aus Buffer lesen *)
		n1 := 0;
		tmp_dw := 0;
		REPEAT
			n2 := MIN(HeaderSize - n1, buf_totalsize - DATA._GetEnd);
			FOR n := 1 TO n2 DO
				tmp_dw := ROL(tmp_dw,8) OR BYTE_TO_DWORD(data.BUF[DATA._GetEnd]);
				DATA._GetEnd := DATA._GetEnd + 1;
			END_FOR;
			IF DATA._GetEnd >= buf_totalsize THEN
				DATA._GetEnd := 0;
			END_IF
			n1 := n1 + n2;
		UNTIL n1 >= HeaderSize
		END_REPEAT;
	
		DATA._GetStart := DATA._GetEnd;
		cnt := DWORD_TO_UINT(tmp_dw AND 16#0000_FFFF);
		DATA.D_SIZE := cnt;
		DATA.D_HEAD := DWORD_TO_WORD(SHR(tmp_dw,16));
	
		x := WORD_TO_BYTE(DATA.D_HEAD); (* nur rechtes byte auswerten *)
		CASE x OF
		01:	pTmp := ADR(DATA.D_STRING); (* String verarbeiten *)
		02:	pTmp := ADR(DATA.D_REAL); (* Real verarbeiten *)
		03:	pTmp := ADR(DATA.D_DWORD); (* DWORD verarbeiten *)
		END_CASE;
	
		(* Daten aus Buffer lesen *)
		n1 := 0;
		REPEAT
			n2 := MIN(cnt - n1, buf_totalsize - DATA._GetEnd);
			FOR n := 1 TO n2 DO
				pTmp^ := data.BUF[DATA._GetEnd];
				pTmp := pTmp + 1;
				DATA._GetEnd := DATA._GetEnd + 1;
			END_FOR;
			IF DATA._GetEnd >= buf_totalsize THEN
				DATA._GetEnd := 0;
			END_IF
			n1 := n1 + n2;
		UNTIL n1 >= cnt
		END_REPEAT;
		IF x = 1 THEN
			pTmp^ := 0; (* String terminieren *)
		END_IF;
		DATA.D_MODE := 0;
	
		(*####################  DEBUG-MESSAGE  ###################################*)
		(*IF _debug_enable THEN
			LOG_CL.NEW_MSG := 'RP: READ /HEAD ~1 / SIZE ~2 / CNT ~3 / >~4<';
			LOG_CL.PRINTF[1] := DWORD_TO_STRH(DATA.D_HEAD);
			LOG_CL.PRINTF[2] := UINT_TO_STRING(cnt);
			LOG_CL.PRINTF[3] := UINT_TO_STRING(DATA.BUF_COUNT);
			CASE x OF
			01:	LOG_CL.PRINTF[4] := DATA.D_STRING;
			02:	LOG_CL.PRINTF[4] := REAL_TO_STRING(DATA.D_REAL);
			03:	LOG_CL.PRINTF[4] := DWORD_TO_STRH(DATA.D_DWORD);
			ELSE
				LOG_CL.PRINTF[4] := '';
			END_CASE;
			LOG_MSG();
		END_IF;*)
		(*########################################################################*)
	END_IF;

	IF (mode_last = 10 AND DATA.D_MODE = 11) OR (mode_last = 12 AND DATA.D_MODE = 0) THEN (* löschen nur direkt nach lesen möglich *)
		mode_last := DATA.D_MODE;
		DATA.BUF_SIZE := DATA.BUF_SIZE - cnt - HeaderSize;
		DATA.BUF_COUNT := DATA.BUF_COUNT - 1;
		DATA._First := DATA._GetEnd;
		DATA.BUF_USED := UINT_TO_USINT(100 * DATA.BUF_SIZE / SIZEOF(DATA.BUF)); (* benützer Speicher in % *)
		DATA.D_MODE := 0;

		(*####################  DEBUG-MESSAGE  ###################################*)
		(*IF _debug_enable THEN
			LOG_CL.NEW_MSG := 'RP: DEL /HEAD ~1 / SIZE ~2 / CNT ~3 / >~4<';
			LOG_CL.PRINTF[1] := DWORD_TO_STRH(DATA.D_HEAD);
			LOG_CL.PRINTF[2] := UINT_TO_STRING(cnt);
			LOG_CL.PRINTF[3] := UINT_TO_STRING(DATA.BUF_COUNT);
			CASE x OF
			01:	LOG_CL.PRINTF[4] := DATA.D_STRING;
			02:	LOG_CL.PRINTF[4] := REAL_TO_STRING(DATA.D_REAL);
			03:	LOG_CL.PRINTF[4] := DWORD_TO_STRH(DATA.D_DWORD);
			ELSE
				LOG_CL.PRINTF[4] := '';
			END_CASE;
			LOG_MSG();
		END_IF;*)
		(*########################################################################*)
	END_IF;

99:	(* Buffer reset - alles löschen *)
	DATA._First := 0;
	DATA._Last := 0;
	DATA._GetStart := 0;
	DATA._GetEnd := 0;
	DATA.BUF_COUNT := 0;
	DATA.BUF_SIZE := 0;
	DATA.BUF_USED := 0;
	DATA.D_STRING := '';
	DATA.D_DWORD := 0;
	DATA.D_REAL := 0.0;
	DATA.D_HEAD := 0;
	DATA.D_MODE := 0;
	DATA.D_SIZE := 0;
	mode_last := 0;
END_CASE;

(* höchsten Auslastungswert speichern *)
IF DATA.BUF_USED > DATA.BUF_USED_MAX THEN
	DATA.BUF_USED_MAX := DATA.BUF_USED;
END_IF;

(* revision history
ks	01. jan. 2011	rev 1.0
	original version
ks	25. jul. 2011	rev 1.1
	neuen MODE 12 hinzugefügt
ks	03. Sep. 2015	rev 1.2
	Auslastungsüberwachung hinzugefügt
ks	21. mar. 2016	rev 1.3
	D_SIZE info hinzugefügt
	Buffer size auf 8192 vergroessert
*)

END_FUNCTION_BLOCK

// POUs/DATA_LOG/DLOG_CRON_TAB
FUNCTION_BLOCK DLOG_CRON_TAB
VAR_INPUT
	ACTIVATE : BOOL;
	DTI : DT;
	SECOND : STRING(20);
	MINUTE : STRING(20);
	HOUR : STRING(20);
	DAY_OF_MONTH : STRING(20);
	DAY_OF_WEEK : STRING(20);
	MONTH : STRING(20);
END_VAR
VAR_OUTPUT
	Q : BOOL;
END_VAR
VAR
	CD :  DLOG_CRON_DATA;
	activate_old : BOOL;
	datei : DATE;
	dti_last : DT;
	cnt1 : INT;
	cnt2 : INT;
	idx1 : INT;
	idx2 : INT;
	idx3 : INT;
	idx4 : INT;
	pos1 : INT;
	pos2 : INT;
	char_cnt : INT;
	trig_day : BOOL;
	trig_weekday : BOOL;
	str1 : STRING(OSCAT_BASIC.STRING_LENGTH);
	str2 : STRING(OSCAT_BASIC.STRING_LENGTH);
	str3 : STRING(OSCAT_BASIC.STRING_LENGTH);
	num_str1 : STRING(10);
END_VAR

(*
version 1.0		27. oct. 2012
programmer		ks
tested by			ks

DLOG_CRON_TAB erzeugt eine Zeit/Datum Tabelle um damit Ein/Ausschaltvorgänge vorzunehmen
*)

IF ACTIVATE THEN
	IF NOT activate_old THEN
		CD.CE[0].VALUE_MIN := 0;	(* Sekunden *)
		CD.CE[0].VALUE_MAX := 59;
		CD.CE[1].VALUE_MIN := 0;	(* Minuten *)
		CD.CE[1].VALUE_MAX := 59;
		CD.CE[2].VALUE_MIN := 0;	(* Stunden *)
		CD.CE[2].VALUE_MAX := 59;
		CD.CE[3].VALUE_MIN := 1;	(* Tage *)
		CD.CE[3].VALUE_MAX := 31;
		CD.CE[4].VALUE_MIN := 1;	(* Wochentag *)
		CD.CE[4].VALUE_MAX := 7;
		CD.CE[5].VALUE_MIN := 1;	(* Monat *)
		CD.CE[5].VALUE_MAX := 12;

		FOR idx1 := 0 TO 5 DO
			idx3 := CD.CE[idx1].VALUE_MIN;
			idx4 := CD.CE[idx1].VALUE_MAx;
			FOR idx2 := idx3 TO idx4 DO
				CD.CE[idx1].ELEMENTS[idx2] := FALSE;
			END_FOR;
			CD.CE[idx1].ALL_SELECTED := FALSE;
		END_FOR;

		str1 := CONCAT(SECOND,'#');
		str1 := CONCAT(str1,MINUTE);
		str1 := CONCAT(str1,'#');
		str1 := CONCAT(str1,HOUR);
		str1 := CONCAT(str1,'#');
		str1 := CONCAT(str1,DAY_OF_MONTH);
		str1 := CONCAT(str1,'#');
		str1 := CONCAT(str1,DAY_OF_WEEK);
		str1 := CONCAT(str1,'#');
		str1 := CONCAT(str1,MONTH);

		FOR idx1 := 0 TO 5 DO
			str2 := ELEMENT_GET(BYTE#35, idx1, str1);
			IF LEN(str2) > 0 THEN
				cnt1 := ELEMENT_COUNT(BYTE#44, str2);	(* Trenzeichen ',' *)
			ELSE
				cnt1 := 1;
			END_IF;

			FOR idx2 := 0 TO cnt1 -1 DO
				str3 := ELEMENT_GET(BYTE#44, idx2, str2);
				IF FIND(str3, '*/') > 0 AND LEN(str3) <= 10 THEN
					pos1 := OSCAT_BASIC.DEC_TO_INT(str3);
					IF pos1 > 0 THEN
						idx3 := CD.CE[idx1].VALUE_MIN;
						idx4 := CD.CE[idx1].VALUE_MAX;
						WHILE idx3 <= idx4 DO
							CD.CE[idx1].ELEMENTS[idx3] := TRUE;
							idx3 := idx3 + pos1;
						END_WHILE;
					END_IF;

				ELSE
					IF FIND(str3, '*') > 0 OR LEN(str3) = 0 THEN
						pos1 := CD.CE[idx1].VALUE_MIN;
						pos2 := CD.CE[idx1].VALUE_MAX;
						CD.CE[idx1].ALL_SELECTED := TRUE;
					ELSE
						cnt2 := ELEMENT_COUNT(BYTE#45, str3);	(* Trenzeichen '-' *)
						char_cnt := LEN(str3);
						IF char_cnt >= 1 AND char_cnt <= 10 THEN
							num_str1 := ELEMENT_GET(BYTE#45, 0, str3);
							pos1 := OSCAT_BASIC.DEC_TO_INT(num_str1);
							pos2 := pos1;
							IF cnt2 = 2 THEN
								num_str1 := ELEMENT_GET(BYTE#45, 1, str3);
								pos2 := OSCAT_BASIC.DEC_TO_INT(num_str1);
							END_IF;
						END_IF;
					END_IF;

					IF pos1 >= CD.CE[idx1].VALUE_MIN AND pos2 <= CD.CE[idx1].VALUE_MAX THEN
						FOR idx3 := pos1 TO pos2 DO
							CD.CE[idx1].ELEMENTS[idx3] := TRUE;
						END_FOR;
					END_IF;
				END_IF;
			END_FOR;
		END_FOR;
	ELSIF DTI <> dti_last THEN
		CD.CE[0].VALUE := OSCAT_BASIC.SECOND_OF_DT(DTI); (* Sekunden *)
		CD.CE[1].VALUE := OSCAT_BASIC.MINUTE_OF_DT(DTI); (* Minuten *)
		CD.CE[2].VALUE := OSCAT_BASIC.HOUR_OF_DT(DTI); (* Stunden *)
		datei := DT_TO_DATE(DTI);
		CD.CE[3].VALUE := OSCAT_BASIC.DAY_OF_MONTH(datei); (* Tag *)
		CD.CE[4].VALUE := OSCAT_BASIC.DAY_OF_WEEK(datei); (* Wochentag *)
		CD.CE[5].VALUE := OSCAT_BASIC.MONTH_OF_DATE(datei); (*  Monat *)
		dti_last := DTI;

		idx2 := CD.CE[0].VALUE;	(* sekunden *)
		Q := CD.CE[0].ELEMENTS[idx2] = TRUE;
		idx2 := CD.CE[1].VALUE;	(* minuten *)
		Q := Q AND CD.CE[1].ELEMENTS[idx2] = TRUE;
		idx2 := CD.CE[2].VALUE;	(* stunden *)
		Q := Q AND CD.CE[2].ELEMENTS[idx2] = TRUE;
		idx2 := CD.CE[5].VALUE;	(* monat *)
		Q := Q AND CD.CE[5].ELEMENTS[idx2] = TRUE;

		(* auswertung Tag und Wochentag *)
		idx2 := CD.CE[3].VALUE;	(* Tag *)
		trig_day:= CD.CE[3].ELEMENTS[idx2] = TRUE;
		idx2 := CD.CE[4].VALUE;	(* Wochentag *)
		trig_weekday := CD.CE[4].ELEMENTS[idx2] = TRUE;

		IF CD.CE[3].ALL_SELECTED = FALSE AND CD.CE[4].ALL_SELECTED = TRUE THEN
			Q := Q AND trig_day; (* nur Tag auswerten *)
		ELSIF CD.CE[3].ALL_SELECTED = TRUE AND CD.CE[4].ALL_SELECTED = FALSE THEN
			Q := Q AND trig_weekday; (* nur Wochentag auswerten *)
		ELSIF CD.CE[3].ALL_SELECTED = FALSE AND CD.CE[4].ALL_SELECTED = FALSE THEN
			Q := Q AND (trig_weekday OR trig_day); (* Tag und Wochentag auswerten *)
		END_IF;
	END_IF;

END_IF;
activate_old := ACTIVATE;

(* revision history
ks	27. oct. 2011	rev 1.0
	original version
*)

END_FUNCTION_BLOCK

// POUs/OTHER/ELEMENT_GET
FUNCTION ELEMENT_GET : STRING(ELEMENT_LENGTH)
VAR_INPUT
	SEP : BYTE;
	POS : INT;
END_VAR
VAR_IN_OUT
	ELEMENT : STRING(ELEMENT_LENGTH);
END_VAR
VAR
	i : INT := 1;
	o : INT := 1;
	pt : POINTER TO ARRAY[1..ELEMENT_LENGTH] OF BYTE;
	po : POINTER TO ARRAY[1..ELEMENT_LENGTH] OF BYTE;
	cnt: INT;
	c: BYTE;
END_VAR

(*
version 1.0	05. apr. 2011
programmer 	ks
tested by		kst

ELEMENT_GET liefert das element an der stelle pos einer liste.
die liste liegt als string von elementen vor die mit den zeichen SEP separiert sind.

*)

(* load pointers *)
pt := ADR(ELEMENT);
po := ADR(ELEMENT_GET);

(* search for the n-th occurence of a separation character and store position in i *)
WHILE (cnt < pos) AND (i < ELEMENT_LENGTH) AND (pt^[i] > 0) DO
	IF pt^[i] = sep THEN cnt := cnt + 1; END_IF;
	i := i + 1;
END_WHILE;

(* copy the list element to output *)
IF i < ELEMENT_LENGTH THEN c := pt^[i]; END_IF;
WHILE (c <> sep) AND (c > 0) AND (o < ELEMENT_LENGTH) AND (i < ELEMENT_LENGTH) DO
	po^[o] :=pt^[i];
	o := o + 1;
	i := i + 1;
	c := pt^[i];
END_WHILE;

(* terminate the output string *)
po^[o] := 0;

(* revision histroy
ks 05. apr. 2011	rev 1.0
	original release

*)

END_FUNCTION

// POUs/OTHER/ELEMENT_COUNT
FUNCTION ELEMENT_COUNT : INT
VAR_INPUT
	SEP : BYTE;
END_VAR
VAR_IN_OUT
	ELEMENT : STRING(ELEMENT_LENGTH);
END_VAR
VAR
	pt : POINTER TO ARRAY[1..ELEMENT_LENGTH] OF BYTE;
	l: INT;
	pos: INT;
END_VAR

(*
version 1.0	05. apr. 2011
programmer 	hugo
tested by		oscat

ELEMENT_COUNT liefert die anzahl der elemente einer liste.
die liste liegt als string von elementen vor die mit den zeichen SEP separiert sind.

*)

IF ELEMENT = '' THEN
	ELEMENT_COUNT := 0;
ELSE
	PT := ADR(ELEMENT);
	ELEMENT_COUNT := 1;
	l := LEN(ELEMENT);
	FOR pos := 1 TO l DO
		IF pt^[pos] = SEP THEN ELEMENT_COUNT := ELEMENT_COUNT + 1; END_IF;
	END_FOR;
END_IF;

(* revision histroy
ks	5. apr. 2011	rev 1.0
	original release

*)

END_FUNCTION

// POUs/DATA_LOG/DLOG_DINT
FUNCTION_BLOCK DLOG_DINT
VAR_IN_OUT
	X : DLOG_DATA;
END_VAR
VAR_INPUT
	VALUE : DINT;
	COLUMN : STRING(40);
	DELTA : DINT;
END_VAR
VAR
	UCB : UNI_CIRCULAR_BUFFER;
	id : WORD;
	delta_last : DINT;
	value_last : DINT;
END_VAR

(*
version 1.3		19. apr. 2012
programmer		ks
tested by		ks

DLOG_DINT legt den DINT-Wert als STRING im FIFO-RING-Buffer ab um diesen mit den Baustein DLOG_STORE_* aufzuzeichnen
*)

CASE x.ADD_COM OF

01:	(* ADD INFO *)
	X.ID_MAX := X.ID_MAX + USINT#1;
	id := WORD#16#0801; (* Quelltype DINT , Zieltype STRING *)
02:	(* ADD HEADER *)
	X.UCB.D_STRING := COLUMN;
	X.UCB.D_HEAD := id;
	X.UCB.D_MODE := 1;
	UCB(DATA:=X.UCB); (* Daten eintragen *)
03:	(* ADD DATA *)
	X.UCB.D_STRING := DINT_TO_STRING(value_last);
	X.UCB.D_HEAD := id;
	X.UCB.D_MODE := 1;
	UCB(DATA:=X.UCB); (* Daten eintragen *)
	delta_last := value_last;
04:	(* ADD DATA REQ *)
	IF DELTA <> DINT#0 THEN
		IF VALUE <= (delta_last - DELTA) OR VALUE >= (delta_last + DELTA) THEN
			X.ADD_DATA_REQ := TRUE;
			delta_last := VALUE;
		END_IF;
	END_IF;
END_CASE;
value_last := VALUE;

(* revision history
ks	01. jan. 2011	rev 1.0
	original version

ks	17. may. 2011	rev 1.1
	DELTA Funktion integriert

ks	25. july.   2011	rev 1.2
	neue head information

ks	19. apr.   2012	rev 1.2
	code neu überarbeitet
*)

END_FUNCTION_BLOCK

// POUs/DATA_LOG/DLOG_DT
FUNCTION_BLOCK DLOG_DT
VAR_IN_OUT
	X : DLOG_DATA;
END_VAR
VAR_INPUT
	FMT : STRING := '#A-#D-#H #N:#R:#T';
	COLUMN : STRING(40);
	DELTA : UDINT;
END_VAR

VAR_OUTPUT
END_VAR
VAR
	UCB : UNI_CIRCULAR_BUFFER;
	id : WORD;
	delta_last : DT;
END_VAR

(*
version 1.3		19. apr. 2012
programmer		ks
tested by		ks

DLOG_DT legt den formatierten DT String im FIFO-RING-Buffer ab um diesen mit den Baustein DLOG_STORE_*  aufzuzeichnen
*)

CASE x.ADD_COM OF

01:	(* ADD INFO *)
	X.ID_MAX := X.ID_MAX + USINT#1;
	id := WORD#16#0D01; (* Quelltype DT , Zieltype STRING *)
02:	(* ADD HEADER *)
	X.UCB.D_STRING := COLUMN;
	X.UCB.D_HEAD := id;
	X.UCB.D_MODE := 1;
	UCB(DATA:=X.UCB); (* Daten eintragen *)
03:	(* ADD DATA *)
	X.UCB.D_STRING := OSCAT_BASIC.DT_TO_STRF(DTI:=X.DTI,MS:=0,FMT:=FMT,LANG:=0);
	X.UCB.D_HEAD := id;
	X.UCB.D_MODE := 1;
	UCB(DATA:=X.UCB); (* Daten eintragen *)
	delta_last := X.DTI;
04:	(* ADD DATA REQ *)
	IF DELTA <> UDINT#0 THEN
		IF DT_TO_UDINT(X.DTI) >= (DT_TO_UDINT(delta_last) + DELTA) THEN
			X.ADD_DATA_REQ := TRUE;
			delta_last := X.DTI;
		END_IF;
	END_IF;
END_CASE;

(* revision history
ks	01. jan. 2011	rev 1.0
	original version

ks	17. may. 2011	rev 1.1
	COLUMN STRING(40), delta

ks	25. july.   2011	rev 1.2
	neue head information

ks	19. apr.   2012	rev 1.3
	code neu überarbeitet
*)

END_FUNCTION_BLOCK

// POUs/DEMO/DLOG_FILE_CSV_DEMO
PROGRAM DLOG_FILE_CSV_DEMO
VAR
	cur_dt: DT;
	enable: BOOL := TRUE;
	trig_t : TIME := T#5s;
	trig_m : BOOL;
	error_c: DWORD;
	error_t: BYTE;
	auto_close: TIME := T#10s;

	x1: DLOG_DT;
	x2 : DLOG_REAL;
	x3 : DLOG_DINT;
	x4 : DLOG_BOOL;
	x5: DLOG_STRING;
	x : DLOG_DATA;
	RTC_2: oscat_basic.RTC_2;
	DLOG_STORE_FILE_CSV : DLOG_STORE_FILE_CSV;
	GEN_SIN_1: oscat_basic.GEN_SIN;
	COUNT_DR: oscat_basic.COUNT_DR;
END_VAR

VAR RETAIN
	save_data : DLOG_SAVE;
END_VAR
VAR // added by the converter: edge detectors and wires of the graphical bodies
    _w1 : ANY;
END_VAR

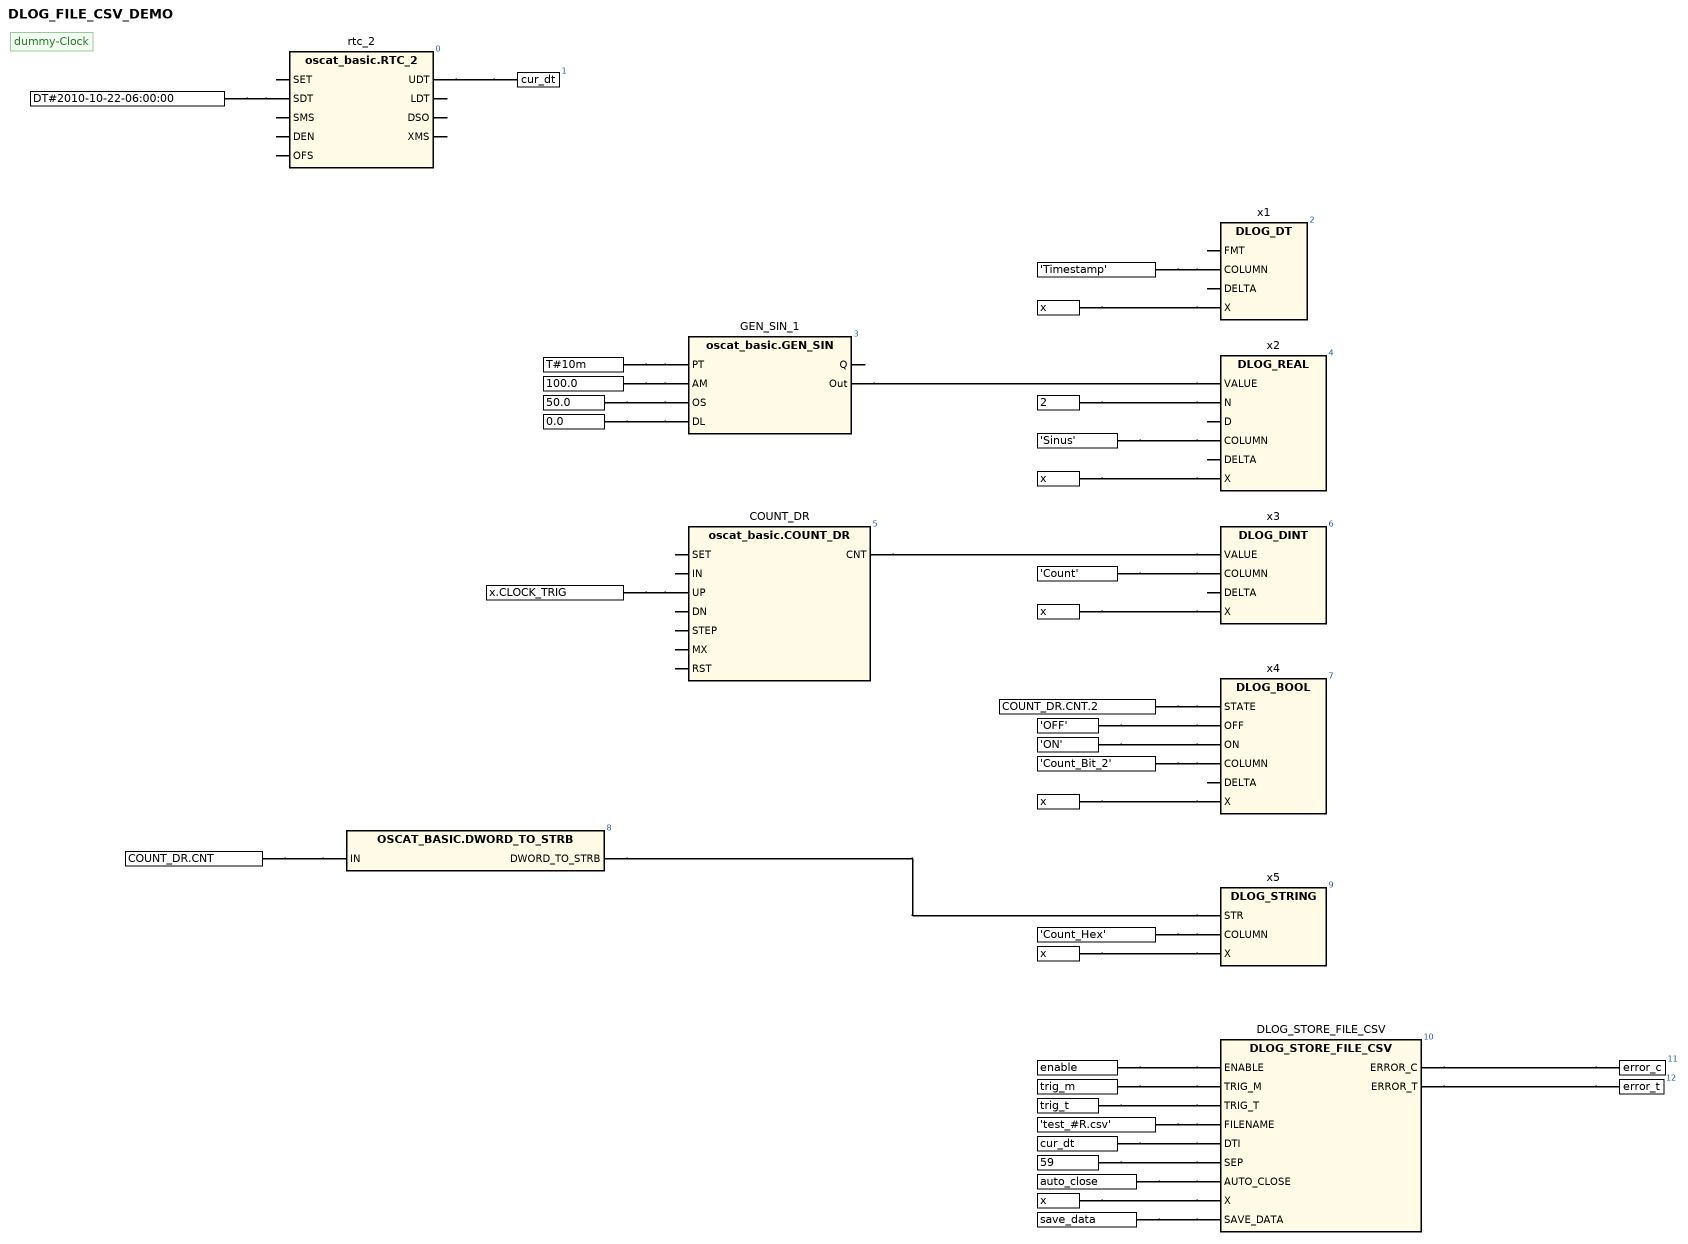
// dummy-Clock
rtc_2(SDT := DT#2010-10-22-06:00:00); // oscat_basic.RTC_2
cur_dt := rtc_2.UDT;
x1(COLUMN := 'Timestamp', X := x); // DLOG_DT
GEN_SIN_1(PT := T#10m, AM := 100.0, OS := 50.0, DL := 0.0); // oscat_basic.GEN_SIN
x2(VALUE := GEN_SIN_1.Out, N := 2, COLUMN := 'Sinus', X := x); // DLOG_REAL
COUNT_DR(UP := x.CLOCK_TRIG); // oscat_basic.COUNT_DR
x3(VALUE := COUNT_DR.CNT, COLUMN := 'Count', X := x); // DLOG_DINT
x4(STATE := COUNT_DR.CNT.2, OFF := 'OFF', ON := 'ON', COLUMN := 'Count_Bit_2', X := x); // DLOG_BOOL
_w1 := OSCAT_BASIC.DWORD_TO_STRB(IN := COUNT_DR.CNT);
x5(STR := _w1, COLUMN := 'Count_Hex', X := x); // DLOG_STRING
DLOG_STORE_FILE_CSV(
    ENABLE := enable,
    TRIG_M := trig_m,
    TRIG_T := trig_t,
    FILENAME := 'test_#R.csv',
    DTI := cur_dt,
    SEP := 59,
    AUTO_CLOSE := auto_close,
    X := x,
    SAVE_DATA := save_data);
error_c := DLOG_STORE_FILE_CSV.ERROR_C;
error_t := DLOG_STORE_FILE_CSV.ERROR_T;

END_PROGRAM

// POUs/DATA_LOG/DLOG_REAL
FUNCTION_BLOCK DLOG_REAL
VAR_IN_OUT
	X : DLOG_DATA;
END_VAR
VAR_INPUT
	VALUE : REAL;
	N : INT;
	D : STRING(1) := ',';
	COLUMN : STRING(40);
	DELTA : REAL;
END_VAR
VAR
	UCB : UNI_CIRCULAR_BUFFER;
	id : WORD;
	delta_last : REAL;
	value_last : REAL;
END_VAR

(*
version 1.3		19. apr. 2012
programmer		ks
tested by		ks

DLOG_REAL legt den REAL-Wert als STRING im FIFO-RING-Buffer ab um diesen mit den Baustein DLOG_STORE_*  aufzuzeichnen
*)

CASE x.ADD_COM OF

01:	(* ADD INFO *)
	X.ID_MAX := X.ID_MAX + USINT#1;
	id := WORD#16#0201; (* Quelltype REAL , Zieltype STRING *)
02:	(* ADD HEADER *)
	X.UCB.D_STRING := COLUMN;
	X.UCB.D_HEAD := id;
	X.UCB.D_MODE := 1;
	UCB(DATA:=X.UCB); (* Daten eintragen *)
03:	(* ADD DATA *)
	X.UCB.D_STRING := OSCAT_BASIC.REAL_TO_STRF(IN:=value_last,N:=N,D:=D);
	X.UCB.D_HEAD := id;
	X.UCB.D_MODE := 1;
	UCB(DATA:=X.UCB); (* Daten eintragen *)
	delta_last := value_last;
04:	(* ADD DATA REQ *)
	IF DELTA <> 0.0 THEN
		IF VALUE <= (delta_last - DELTA) OR VALUE >= (delta_last + DELTA) THEN
			X.ADD_DATA_REQ := TRUE;
			delta_last := VALUE;
		END_IF;
	END_IF;
END_CASE;
value_last := VALUE;

(* revision history
ks	01. jan. 2011	rev 1.0
	original version

ks	17. may. 2011	rev 1.1
	DELTA Funktion integriert

ks	25. july.   2011	rev 1.2
	neue head information

ks	19. apr.   2012	rev 1.3
	code neu überarbeitet
*)

END_FUNCTION_BLOCK

// POUs/DATA_LOG/DLOG_STRING
FUNCTION_BLOCK DLOG_STRING
VAR_IN_OUT
	X : DLOG_DATA;
END_VAR
VAR_INPUT
	STR : STRING;
	COLUMN : STRING(40);
END_VAR
VAR_OUTPUT
END_VAR
VAR
	UCB : UNI_CIRCULAR_BUFFER;
	id : WORD;
	str_last : STRING;
END_VAR

(*
version 1.3		19. apr. 2012
programmer		ks
tested by		ks

DLOG_STRING legt den STRING im FIFO-RING-Buffer ab um diesen mit den Baustein DLOG_STORE_*  aufzuzeichnen
*)

CASE x.ADD_COM OF

01:	(* ADD INFO *)
	X.ID_MAX := X.ID_MAX + USINT#1;
	id := WORD#16#0101; (* Quelltype STRING , Zieltype STRING *)
02:	(* ADD HEADER *)
	X.UCB.D_STRING := COLUMN;
	X.UCB.D_HEAD := id;
	X.UCB.D_MODE := 1;
	UCB(DATA:=X.UCB); (* Daten eintragen *)
03:	(* ADD DATA *)
	X.UCB.D_STRING := str_last;
	X.UCB.D_HEAD := id;
	X.UCB.D_MODE := 1;
	UCB(DATA:=X.UCB); (* Daten eintragen *)
END_CASE;
str_last := STR;

(* revision history
ks	01. jan. 2011	rev 1.0
	original version

ks	17. may. 2011	rev 1.1
	COLUMN STRING(40)

ks	25. july.   2011	rev 1.2
	neue head information

ks	19. apr.   2012	rev 1.3
	code neu überarbeitet
*)

END_FUNCTION_BLOCK

// POUs/DATA_LOG/DLOG_STORE_FILE_CSV
FUNCTION_BLOCK DLOG_STORE_FILE_CSV
VAR_IN_OUT
	X : DLOG_DATA;
	SAVE_DATA : DLOG_SAVE;
END_VAR
VAR_INPUT
	ENABLE : BOOL;
	TRIG_M : BOOL;
	TRIG_T : TIME;
	FILENAME : STRING;
	DTI : DT;
	SEP : BYTE;
	AUTO_CLOSE : TIME := T#15s;
END_VAR
VAR_OUTPUT
	ERROR_C : DWORD;
	ERROR_T : BYTE;
END_VAR
VAR
	FS : FILE_SERVER;
	FSD : FILE_SERVER_DATA;
	PT : NETWORK_BUFFER;
	UCB : UNI_CIRCULAR_BUFFER;
	trig_auto : BOOL;
	trig_stored : BOOL;
	trig_tmp : BOOL;
	trig_m_last : BOOL;
	dti_last : DT := DT#2070-02-06-06:28:15;
	fn_last : STRING;
	fn : STRING;
	step_1: INT;
	step_2: INT;
	idx : INT;
	log_stop : BOOL;
	n : USINT;
	wd_ton : TON;
	wd_time : TIME;
	aw_ton : TON;
	aw_enable : BOOL;
	aw_aktiv : BOOL;
	total_bytes : UDINT;

	(*
	LOG_MSG : LOG_MSG;
	_debug_enable : BOOL := TRUE;
	*)
END_VAR

(*
version 1.5		21. mar. 2016
programmer		ks
tested by			ks

DLOG_STORE_FILE_CSV der Baustein schreibt die DLOG Parameter in einen lokale Datei im CSV-Format
*)

X.DTI := DTI; (* Datum / Zeit eintragen *)
X.CLOCK_TRIG := DTI <> dti_last;
dti_last := DTI;
trig_auto := FALSE;
IF X.CLOCK_TRIG THEN (* Impuls in jeder Sekunde *)
	fn := OSCAT_BASIC.DT_TO_STRF(DTI, 0, FILENAME, 0); (* automatische Dateinamen generierung *)
	IF TRIG_T >= T#1000ms THEN (* automatischer Trigger *)
		trig_auto := DT_TO_UDINT(DTI) MOD (TIME_TO_UDINT(TRIG_T) / UDINT#1000) = UDINT#0;
	END_IF;
END_IF;

CASE step_1 OF

00:	IF ENABLE THEN
		aw_enable := AUTO_CLOSE >= T#5s;
		wd_time := SEL(X.LOAD_TIME_MAX > T#0s, T#5ms,X.LOAD_TIME_MAX);
		fn_last := fn; (* aktuellen Dateinnamen speichern *)
		IF X.ID_MAX = USINT#0 THEN (* nur einmal nach Satellitenbausteinen scannen *)
			X.ADD_COM := 01; (* ADD INFO *)
			X.STORE_TYPE := BYTE#2; (* CSV-Modus *)
		END_IF;
		step_1 := 10;

		(* ---------------- Debug-Message -----------------------*)
		(*IF _debug_enable THEN
			LOG_CL.NEW_MSG := 'FILE_CSV1 - Start: File [~1], [~2]';
			LOG_CL.PRINTF[1] := fn_last;
			LOG_CL.PRINTF[2] := DT_TO_STRING(DTI);
			LOG_MSG();
		END_IF;*)
		(* -----------------------------------------------------------------*)

	END_IF;

10:	X.UCB.D_STRING := fn_last;
	IF fn_last = SAVE_DATA.FN_REM THEN
		X.UCB.D_HEAD := WORD#16#F201; (* Filemode open + write *)
		X.ADD_COM := 00;
	ELSE
		X.UCB.D_HEAD := WORD#16#F301; (* Filemode create + write *)
		X.ADD_COM := 02; (* ADD HEADER *)
	END_IF;

	X.UCB.D_MODE := 1; (* Dateinamen als String ablegen *)
	UCB(DATA:=X.UCB); (* Daten eintragen *)
	step_1 := 30;

30:	(* LOG-Trigger verarbeiten *)
	trig_tmp := (TRIG_M AND NOT trig_m_last) OR trig_auto OR X.ADD_DATA_REQ;

	IF ENABLE = FALSE OR fn <> fn_last THEN (* ENABLE = 0 oder neuen Dateinamen -> Log Stop *)
		trig_stored := trig_tmp; (* aktuellen Triggerpuls speichern *)
		X.UCB.D_HEAD := WORD#16#EE00;
		X.UCB.D_MODE := 1;
		UCB(DATA:=X.UCB); (* Element schreiben *)
		X.ADD_COM := 00;
		step_1 := 00;

		(* ---------------- Debug-Message -----------------------*)
		(*IF _debug_enable THEN
			LOG_CL.NEW_MSG := 'FILE_CSV1 - Stop: [~2]';
			LOG_CL.PRINTF[2] := DT_TO_STRING(DTI);
			LOG_MSG();
		END_IF;*)
		(* -----------------------------------------------------------------*)

	ELSIF ENABLE THEN
		IF trig_tmp OR trig_stored THEN (* manueller, automatischer oder externer Trigger *)
			trig_stored := FALSE;
			X.ADD_COM := 03; (* ADD DATA *)
			SAVE_DATA.TRIG_CNT := SAVE_DATA.TRIG_CNT + UDINT#1;
			SAVE_DATA.TRIG_CNT_TOTAL  := SAVE_DATA.TRIG_CNT_TOTAL + UDINT#1;
			(* ---------------- Debug-Message -----------------------*)
			(*IF _debug_enable THEN
				LOG_CL.NEW_MSG := 'FILE_CSV1 - Trig: [~2]';
				LOG_CL.PRINTF[2] := DT_TO_STRING(DTI);
				LOG_MSG();
			END_IF;*)
			(* -----------------------------------------------------------------*)
		ELSE
			X.ADD_COM := 04;	(* ADD DATA REQ *)
		END_IF;
	END_IF;

END_CASE;
X.ADD_DATA_REQ := FALSE; (* externe Anforderung rücksetzen *)

(* ##################################### *)

CASE step_2 OF

00:	aw_ton(IN:= idx > 0 AND aw_enable, PT:= AUTO_CLOSE); (* AutoWrite Timer *)
	IF aw_ton.Q THEN (* Zeitgesteuertes Datenschreiben *)
		aw_aktiv := TRUE;
		step_2 := 10; (* Daten schreiben *)
		(* ---------------- Debug-Message -----------------------*)
		(*IF _debug_enable THEN
			LOG_CL.NEW_MSG := 'FILE_CSV2 - AutoWrite: [~2]';
			LOG_CL.PRINTF[2] := DT_TO_STRING(DTI);
			LOG_MSG();
		END_IF;*)
		(* -----------------------------------------------------------------*)

	ELSE
		wd_ton(IN:= FALSE, PT:= wd_time);
		wd_ton(IN:= TRUE);
		WHILE X.UCB.BUF_COUNT > 0 AND step_2 = 0 AND wd_ton.Q = FALSE DO

			X.UCB.D_MODE := 10;
			UCB(DATA:=X.UCB); (* Element lesen , aber noch nicht entfernen *)
			IF X.UCB.D_HEAD > WORD#16#F000 THEN (* F301 oder F201 *)
				X.UCB.D_MODE := 11;
				UCB(DATA:=X.UCB); (* Element entfernen *)
	
				FSD.MODE := WORD_TO_BYTE(SHR(SHL(X.UCB.D_HEAD,4),12)); (* 0X00 -> 000X = 3 create + write / 2 open + write *)
				FSD.OFFSET := UDINT#0; (* Start bei Dateianfang *)
				FSD.FILENAME := X.UCB.D_STRING; (* Dateiname *)
				PT.SIZE := UINT#0;
				SAVE_DATA.FN_REM := FSD.FILENAME; (* aktuellen Dateinamen remanent sichern *)
	
				IF FSD.MODE = BYTE#3 THEN	(* Datei neu anlegen -> dann zähler reset *)
					SAVE_DATA.TRIG_CNT := UDINT#0;
				END_IF;
	
				X.NEW_FILE := FSD.FILENAME;
				X.NEW_FILE_SIZE := UDINT#0;
				X.NEW_FILE_RTRIG := FALSE;
				step_2 := 20;
				(* ---------------- Debug-Message -----------------------*)
				(*IF _debug_enable THEN
					LOG_CL.NEW_MSG := 'FILE_CSV2 - Create: Mode [~1] , [~2]';
					LOG_CL.PRINTF[2] := DT_TO_STRING(DTI);
					LOG_CL.PRINTF[1] := BYTE_TO_STRING(FSD.MODE);
					LOG_MSG();
				END_IF;*)
				(* -----------------------------------------------------------------*)

			ELSIF X.UCB.D_HEAD = WORD#16#EE00 THEN (* LOG_STOP Command *)
				X.UCB.D_MODE := 11;
				UCB(DATA:=X.UCB); (* Element entfernen *)
				log_stop := TRUE;
				step_2 := 10; (* Daten schreiben *)

			ELSIF idx + X.UCB.D_SIZE + 2 < SIZEOF(PT.BUFFER) THEN (* bufferplatz vorhanden *)
				X.UCB.D_MODE := 11;
				UCB(DATA:=X.UCB); (* Element entfernen *)
				(* ---------------- Debug-Message -----------------------*)
				(*IF _debug_enable THEN
					LOG_CL.NEW_MSG := 'FILE_CSV2 - BUF: TXT [~1],Pos [~2], [~3]';
					LOG_CL.PRINTF[1] := X.UCB.D_STRING;
					LOG_CL.PRINTF[2] := INT_TO_STRING(idx);
					LOG_CL.PRINTF[3] := DT_TO_STRING(DTI);
					LOG_MSG();
				END_IF;*)
				(* -----------------------------------------------------------------*)
				OSCAT_BASIC._STRING_TO_BUFFER(STR:=X.UCB.D_STRING, POS:=idx, PT:=ADR(PT.BUFFER), SIZE:=SIZEOF(PT.BUFFER));
				idx := idx + LEN(X.UCB.D_STRING);
				n := n + USINT#1;
				IF n = X.ID_MAX THEN (* letztes Element einer Zeile *)
					n := USINT#0;
					PT.BUFFER[idx] := BYTE#16#0D;
					idx := idx + 1;
					PT.BUFFER[idx] := BYTE#16#0A;
				ELSE
					PT.BUFFER[idx] := SEP;
				END_IF;
				idx := idx + 1;
				X.NEW_FILE_SIZE := total_bytes + INT_TO_UDINT(idx);
			ELSE (* kein Platz vorhanden *)
				step_2 := 10; (* Daten schreiben *)
			END_IF;
			wd_ton();
		END_WHILE;
	END_IF;

10:	IF idx > 0 THEN (* Daten schreiben *)
		FSD.MODE := BYTE#2; (* File_Open_Exist + File_Write *)
		FSD.OFFSET := UDINT#4294967294; (* 16#FFFF_FFFE ->Spezialcode: Daten automatisch an Dateiende anhängen *)
		PT.SIZE := INT_TO_UINT(idx); (* Datenlänge eintragen *)
		idx := 0;
		(* ---------------- Debug-Message -----------------------*)
		(*IF _debug_enable THEN
			LOG_CL.NEW_MSG := 'FILE_CSV2 - WriteData: Mode [~3] Size [~1] , [~2]';
			LOG_CL.PRINTF[1] := UINT_TO_STRING(PT.SIZE);
			LOG_CL.PRINTF[2] := DT_TO_STRING(DTI);
			LOG_CL.PRINTF[3] := BYTE_TO_STRING(FSD.MODE);
			LOG_MSG();
		END_IF;*)
		(* -----------------------------------------------------------------*)
	END_IF;
	step_2 := 20;

20:	IF FSD.MODE = BYTE#0 THEN
		total_bytes := FSD.FILE_SIZE;
		X.NEW_FILE_SIZE := total_bytes + INT_TO_UDINT(idx);
		IF log_stop OR aw_aktiv THEN
			aw_aktiv := FALSE;
			FSD.MODE := BYTE#5; (* Datei schliessen *)
			(* ---------------- Debug-Message -----------------------*)
			(*IF _debug_enable THEN
				LOG_CL.NEW_MSG := 'FILE_CSV2 - Close: [~2]';
				LOG_CL.PRINTF[2] := DT_TO_STRING(DTI);
				LOG_MSG();
			END_IF;*)
			(* -----------------------------------------------------------------*)
		END_IF;
		step_2 := 30;
	END_IF;

30:	IF FSD.MODE = BYTE#0 THEN (* Befehl beendet ? *)
		IF log_stop THEN
			X.NEW_FILE_RTRIG := TRUE;
			log_stop := FALSE;
			SAVE_DATA.FN_REM := ''; (* remanenten Dateinamen löschen *)
		END_IF;
		step_2 := 00;
	END_IF;

END_CASE;

